REGION Network 7: GlueCalibratonMode Manual Mode Reset Test
   RUNG wire#powerrail
      Contact( "Station_Sys".Manual.Mode )
      Contact( "GluingControl".GlueCalibratonMode )
      Contact( "GluingControl".Control.ManualTest_X )
      Contact( "IAI_DeviceCtl".IAIServo[2].Point[1].Achieve )
      Contact( "IAI_DeviceCtl".IAIServo[1].Point[1].Achieve )
      Contact( "IAI_DeviceCtl".IAIServo[3].Point[1].Achieve )
      { S7_Templates := "time_type := LTime" } "GluingControl".TON[1].TONR(r := wire#w2, pt := LT#10.7S, et =>)
   END_RUNG
   RUNG wire#powerrail
      Contact( "GluingControl".GlueCalibratonMode )
      wire#w1
      P_Trig( "GluingControl".P[1] )
   END_RUNG wire#w2
   RUNG wire#powerrail
      I_Contact( "Station_Sys".Manual.Mode )
   END_RUNG wire#w1
   RUNG wire#powerrail
      { S7_Templates := "SrcType := LTime" } EQ_Contact(in1 := "GluingControl".TON[1].ET, in2 := LT#10.7S)
      R_Coil( "GluingControl".Control.ManualTest_X )
      R_Coil( "GluingControl".GlueCalibratonMode )
   END_RUNG
   // the same network as SCL:
   #_w1 := "GluingControl".GlueCalibratonMode OR NOT "Station_Sys".Manual.Mode;
   #_w2 := #_w1 AND NOT "GluingControl".P[1];   // rising edge
   "GluingControl".P[1] := #_w1;
   "GluingControl".TON[1].TONR(IN := "Station_Sys".Manual.Mode AND "GluingControl".GlueCalibratonMode AND "GluingControl".Control.ManualTest_X AND "IAI_DeviceCtl".IAIServo[2].Point[1].Achieve AND "IAI_DeviceCtl".IAIServo[1].Point[1].Achieve AND "IAI_DeviceCtl".IAIServo[3].Point[1].Achieve,
                           R := #_w2,
                           PT := LT#10.7S);
   IF "GluingControl".TON[1].ET = LT#10.7S THEN
       "GluingControl".Control.ManualTest_X := FALSE;
       "GluingControl".GlueCalibratonMode := FALSE;
   END_IF;
END_REGION
END_FUNCTION

FUNCTION "Pallet_NG" : Void   // FC2900, LAD
{ S7_Optimized_Access := 'TRUE' }
// stored: AutoNumber false, SetENOAutomatically false
   VAR_INPUT
      iSysMode : "RCS_SysComInterface_V1";
   END_VAR
BEGIN

REGION Network 1 (SCL): NG BOXES MAIN FUNCTION BLOCK
   "NG_BOXES_DB"(
                 in_Permission_to_Open :=
                 // in manual mode always
                 #iSysMode.ManualMode OR
                 // 
                 (
                 // all 3 robots are in safe step and have no job / no task running
                 "ST10_Flow5_FRobot_1_iDB"."Open NG BOX REQUESTED?".X AND
                 "ST10_Flow8_FRobot_2_iDB"."Open NG BOX REQUESTED?".X AND
                 "ST10_Flow15_FRobot_3_iDB"."Open NG BOX REQUESTED?".X
                 ) OR "Robot_DB".NG_box_open_flag_during_auto
                 );
END_REGION
END_FUNCTION

FUNCTION_BLOCK "NG_BOXES"   // FB3, SCL
{ S7_Optimized_Access := 'TRUE' }
// stored: MemoryReserve 1000, SetENOAutomatically false
   VAR_INPUT
      in_Permission_to_Open : Bool;
   END_VAR
   VAR_OUTPUT
      out_Request_to_open : Bool;
   END_VAR
   VAR
      Box_Loading { S7_SetPoint := 'True'} : "FB_NG_Box_Control";
      Box_Unloading { S7_SetPoint := 'True'} : "FB_NG_Box_Control";
      TempSensors : Array[1..15] of Bool;
   END_VAR
BEGIN
   // ==========================================================================
   // BOX 1: LOADING – MACHINE LOADING SIDE                                   // EN: Loading side of machine (material IN)
   //                                                                          // CN: 机器上料侧（物料进入机器）
   //                                                                          // SK: Nakladacia / vstupná strana stroja
   // ==========================================================================
   #TempSensors[1] := "iE1-UnloadingShaftPressNG_1";   // EN: NG shaft press pos 1   // CN: 轴压装NG位置1   // SK: NG lis hriadeľa poz.1
   #TempSensors[2] := "iE1-UnloadingShaftPressNG_2";   // EN: NG shaft press pos 2   // CN: 轴压装NG位置2   // SK: NG lis hriadeľa poz.2
   #TempSensors[3] := "iE1-UnloadingShaftPressNG_3";   // EN: NG shaft press pos 3   // CN: 轴压装NG位置3   // SK: NG lis hriadeľa poz.3
   #TempSensors[4] := "iE1-UnloadingShaftPressNG_4";   // EN: NG shaft press pos 4   // CN: 轴压装NG位置4   // SK: NG lis hriadeľa poz.4
   #TempSensors[5] := "iE1-UnloadingShaftPressNG_5";   // EN: NG shaft press pos 5   // CN: 轴压装NG位置5   // SK: NG lis hriadeľa poz.5
   #TempSensors[6] := "iE1-UnloadingShaftScanNG_1";    // EN: NG shaft scan pos 1    // CN: 轴扫描NG位置1   // SK: NG sken hriadeľa 1
   #TempSensors[7] := "iE1-UnloadingShaftScanNG_2";    // EN: NG shaft scan pos 2    // CN: 轴扫描NG位置2   // SK: NG sken hriadeľa 2
   #TempSensors[8] := "iE1-UnloadingShaftScanNG_3";    // EN: NG shaft scan pos 3    // CN: 轴扫描NG位置3   // SK: NG sken hriadeľa 3
   #TempSensors[9] := "iE1-UnloadingShaftScanNG_4";    // EN: NG shaft scan pos 4    // CN: 轴扫描NG位置4   // SK: NG sken hriadeľa 4
   #TempSensors[10] := "iE1-UnloadingShaftScanNG_5";    // EN: NG shaft scan pos 5    // CN: 轴扫描NG位置5   // SK: NG sken hriadeľa 5
   #TempSensors[11] := "iE1-UnloadingRingScanNG_1";     // EN: NG ring scan pos 1     // CN: 环扫描NG位置1   // SK: NG sken krúžku 1
   #TempSensors[12] := "iE1-UnloadingRingScanNG_2";     // EN: NG ring scan pos 2     // CN: 环扫描NG位置2   // SK: NG sken krúžku 2
   #TempSensors[13] := "iE1-UnloadingRingScanNG_3";     // EN: NG ring scan pos 3     // CN: 环扫描NG位置3   // SK: NG sken krúžku 3
   #TempSensors[14] := "iE1-UnloadingRingScanNG_4";     // EN: NG ring scan pos 4     // CN: 环扫描NG位置4   // SK: NG sken krúžku 4
   #TempSensors[15] := "iE1-UnloadingRingScanNG_5";     // EN: NG ring scan pos 5     // CN: 环扫描NG位置5   // SK: NG sken krúžku 5

   #Box_Loading(
                Button        := "iNG_Button1",                     // EN: Operator button (loading side)   // CN: 上料侧操作按钮   // SK: Tlačidlo obsluhy – loading
                MagnetSensor  := "iE-NG-01Detection",               // EN: Door closed sensor                // CN: 门关闭传感器     // SK: Snímač zatvorenia dverí
                LockedFB      := NOT "iE-NG-01 Safety Gate_UnLock", // EN: Lock feedback (locked)             // CN: 锁定反馈         // SK: Spätná väzba – zamknuté
                UnlockedFB    := "iE-NG-01 Safety Gate_UnLock",     // EN: Lock feedback (unlocked)           // CN: 解锁反馈         // SK: Spätná väzba – odomknuté
                AtSafePoint   := #in_Permission_to_Open,            // EN: Sequence at safe point (Step 111)  // CN: 序列在安全步骤   // SK: Sekvencia v bezpečnom kroku
                Sensors       := #TempSensors,
                UnlockCmd     => "ST10_NGGate1_DB"."sSafetyGate UnlockRequest", // EN: Unlock command // CN: 解锁命令 // SK: Príkaz na odomknutie
                LockCmd       => "ST10_NGGate1_DB"."sSafetyGate LockRequest",   // EN: Lock command   // CN: 上锁命令 // SK: Príkaz na zamknutie
                CylinderOpen  => "oE-NG-01NGLocationCylinderToHP",   // EN: Cylinder open (home)  // CN: 气缸打开 // SK: Otvoriť valec
                CylinderClose => "oE-NG-01NGLocationCylinderToWP",   // EN: Cylinder close (work) // CN: 气缸关闭 // SK: Zavrieť valec
                ButtonLight => "oNG_Button1"   ,                    // E,N: Button lamp           // CN: 按钮灯   // SK: Svetlo tlačidla
                Ready_1 => "AutoProcessControl".NG_1.Robot1PutPrimit_1   ,         // Status pro robota: Řada 1 (1-5) má místo // 机器人状态：第1排（1-5）有空位
                Ready_2 => "AutoProcessControl".NG_1.Robot1PutPrimit_2,
                Ready_3 => "AutoProcessControl".NG_1.Robot1PutPrimit_3

   );

   // ==========================================================================
   // BOX 2: UNLOADING – MACHINE UNLOADING SIDE                                // EN: Unloading side of machine (material OUT)
   //                                                                          // CN: 机器下料侧（物料离开机器）
   //                                                                          // SK: Vykladacia / výstupná strana stroja
   // ==========================================================================
   #TempSensors[1] := "iE2-UnloadingPressNG_1";          // EN: NG press pos 1   // CN: 压装NG位置1   // SK: NG lis poz.1
   #TempSensors[2] := "iE2-UnloadingPressNG_2";          // EN: NG press pos 2   // CN: 压装NG位置2   // SK: NG lis poz.2
   #TempSensors[3] := "iE2-UnloadingPressNG_3";          // EN: NG press pos 3   // CN: 压装NG位置3   // SK: NG lis poz.3
   #TempSensors[4] := "iE2-UnloadingPressNG_4";          // EN: NG press pos 4   // CN: 压装NG位置4   // SK: NG lis poz.4
   #TempSensors[5] := "iE2-UnloadingPressNG_5";          // EN: NG press pos 5   // CN: 压装NG位置5   // SK: NG lis poz.5
   #TempSensors[6] := "iE2-UnloadingMagentScanNG_1";     // EN: NG magnet scan 1 // CN: 磁体扫描NG1   // SK: NG magnet sken 1
   #TempSensors[7] := "iE2-UnloadingMagentScanNG_2";     // EN: NG magnet scan 2 // CN: 磁体扫描NG2   // SK: NG magnet sken 2
   #TempSensors[8] := "iE2-UnloadingMagentScanNG_3";     // EN: NG magnet scan 3 // CN: 磁体扫描NG3   // SK: NG magnet sken 3
   #TempSensors[9] := "iE2-UnloadingMagentScanNG_4";     // EN: NG magnet scan 4 // CN: 磁体扫描NG4   // SK: NG magnet sken 4
   #TempSensors[10] := "iE2-UnloadingMagentScanNG_5";     // EN: NG magnet scan 5 // CN: 磁体扫描NG5   // SK: NG magnet sken 5
   #TempSensors[11] := "iE2-UnloadingRingScanNG_1";       // EN: NG ring scan 1   // CN: 环扫描NG1     // SK: NG sken krúžku 1
   #TempSensors[12] := "iE2-UnloadingRingScanNG_2";       // EN: NG ring scan 2   // CN: 环扫描NG2     // SK: NG sken krúžku 2
   #TempSensors[13] := "iE2-UnloadingRingScanNG_3";       // EN: NG ring scan 3   // CN: 环扫描NG3     // SK: NG sken krúžku 3
   #TempSensors[14] := "iE2-UnloadingRingScanNG_4";       // EN: NG ring scan 4   // CN: 环扫描NG4     // SK: NG sken krúžku 4
   #TempSensors[15] := "iE2-UnloadingRingScanNG_5";       // EN: NG ring scan 5   // CN: 环扫描NG5     // SK: NG sken krúžku 5

   #Box_Unloading(
                  Button        := "iNG_Button2",                     // EN: Operator button (unloading side) // CN: 下料侧操作按钮 // SK: Tlačidlo obsluhy – unloading
                  MagnetSensor  := "iE-NG-02Detection",               // EN: Door closed sensor               // CN: 门关闭传感器   // SK: Snímač zatvorenia dverí
                  LockedFB      := NOT "iE-NG-02 Safety Gate_UnLock", // EN: Lock feedback (locked)            // CN: 锁定反馈       // SK: Spätná väzba – zamknuté
                  UnlockedFB    := "iE-NG-02 Safety Gate_UnLock",     // EN: Lock feedback (unlocked)          // CN: 解锁反馈       // SK: Spätná väzba – odomknuté
                  AtSafePoint   := #in_Permission_to_Open,
                  Sensors       := #TempSensors,
                  UnlockCmd     => "ST10_NGGate2_DB"."sSafetyGate UnlockRequest",
                  LockCmd       => "ST10_NGGate2_DB"."sSafetyGate LockRequest",
                  CylinderOpen  => "oE-NG-02NGLocationCylinderToHP",
                  CylinderClose => "oE-NG-02NGLocationCylinderToWP",
                  ButtonLight   => "oNG_Button2",
                  Ready_1 => "AutoProcessControl".NG_2.Robot3PutPrimit_1   ,         // Status pro robota: Řada 1 (1-5) má místo // 机器人状态：第1排（1-5）有空位
                  Ready_2 => "AutoProcessControl".NG_2.Robot3PutPrimit_2,
                  Ready_3 => "AutoProcessControl".NG_2.Robot3PutPrimit_3
   );

   // EN: Request pause of main sequence if any side requests opening
   // CN: 任一侧请求开门时，请求暂停主序列
   // SK: Požiadavka na pauzu hlavnej sekvencie, ak ktorákoľvek strana žiada otvorenie
   #out_Request_to_open := #Box_Loading.PauseReq OR #Box_Unloading.PauseReq;
END_FUNCTION_BLOCK

FUNCTION_BLOCK "FB_NG_Box_Control"   // FB5, SCL
{ S7_Optimized_Access := 'TRUE' }
// stored: MemoryReserve 1000, SetENOAutomatically false
   VAR_INPUT
      Button : Bool;
      MagnetSensor : Bool;
      LockedFB : Bool;
      UnlockedFB : Bool;
      AtSafePoint : Bool;
      Sensors : Array[1..15] of Bool;
   END_VAR
   VAR_OUTPUT
      PauseReq : Bool;
      UnlockCmd : Bool;
      LockCmd : Bool;
      CylinderOpen : Bool;
      CylinderClose : Bool;
      ButtonLight : Bool;
      Ready_1 : Bool;
      Ready_2 : Bool;
      Ready_3 : Bool;
      OpenFlag : Bool;
   END_VAR
   VAR
      State : Int := 99;
      BlinkTimer { S7_SetPoint := 'True'} : TON_TIME;
      BlinkBit : Bool;
      i : Int;
      buttontriggered { S7_SetPoint := 'True'} : R_TRIG;
      c : Int;
   END_VAR
BEGIN
   // 1. POSITION CHECK (Ready_1..3) - TRUE = at least one position in the row is FREE
   // 1. KONTROLA POZÍCIÍ – TRUE = aspoň jedna pozícia v rade je VOĽNÁ
   // 1. 位置检测 – TRUE = 该行中至少有一个位置是空的

   // LINE #1  .... 5 POSITIONS
   // EN: Line 1 checks sensors 1–5 (row 1)
   // SK: Riadok 1 kontroluje senzory 1–5 (riadok 1)
   // CN: 第1行检测传感器1–5（第1排）
   #Ready_1 := FALSE;
   FOR #i := 1 TO 5 DO
     IF NOT #Sensors[#i] THEN
       #Ready_1 := TRUE;
     END_IF;
   END_FOR;

   // LINE #2  .... 5 POSITIONS
   // EN: Line 2 checks sensors 6–10 (row 2)
   // SK: Riadok 2 kontroluje senzory 6–10 (riadok 2)
   // CN: 第2行检测传感器6–10（第2排）
   #Ready_2 := FALSE;
   FOR #i := 6 TO 10 DO
     IF NOT #Sensors[#i] THEN
       #Ready_2 := TRUE;
     END_IF;
   END_FOR;

   // LINE #3  .... 5 POSITIONS
   // EN: Line 3 checks sensors 11–15 (row 3)
   // SK: Riadok 3 kontroluje senzory 11–15 (riadok 3)
   // CN: 第3行检测传感器11–15（第3排）
   #Ready_3 := FALSE;
   FOR #i := 11 TO 15 DO
     IF NOT #Sensors[#i] THEN
       #Ready_3 := TRUE;
     END_IF;
   END_FOR;


   // 2. BLINKING / BUTTON FEEDBACK
   // EN: Blink signal taken from system clock (0.4s)
   // SK: Blikanie je odvodené zo systémového hodinového bitu (0,4 s)
   // CN: 闪烁信号来自系统时钟位（0.4秒）
   #BlinkBit := "ClockMemory0.4s";

   // EN: Rising-edge detection of the button
   // SK: Detekcia nábežnej hrany tlačidla
   // CN: 按钮上升沿检测
   #buttontriggered(CLK := #Button);


   // 3. DOOR STATE MACHINE
   // EN: Main state machine controlling door, lock and cylinder
   // SK: Hlavný stavový automat pre dvere, zámok a valec
   // CN: 门、锁和气缸的主状态机
   CASE #State OF

     99: // INITIALIZATION
       // EN: Decision after PLC start
       // SK: Rozhodnutie po štarte PLC
       // CN: PLC 启动后的状态判断
       IF #MagnetSensor AND #LockedFB THEN
         #State := 0;   // EN: Closed & locked → IDLE
         // SK: Zavreté a zamknuté → IDLE
         // CN: 已关闭并锁定 → 空闲状态
       ELSIF #MagnetSensor AND NOT #LockedFB THEN
         #State := 40;  // EN: Closed but unlocked → wait for confirmation
         // SK: Zavreté, ale odomknuté → čakať na potvrdenie
         // CN: 门已关但未上锁 → 等待确认
       ELSE
         #State := 30;  // EN: Door physically open → OPEN state
         // SK: Dvere fyzicky otvorené → OPEN stav
         // CN: 门处于打开状态 → OPEN
       END_IF;

     0:  // IDLE
       // EN: Normal operation, sequence running
       // SK: Normálna prevádzka, sekvencia beží
       // CN: 正常运行，工序执行中
       #PauseReq := FALSE;
       #UnlockCmd := FALSE;
       #LockCmd := TRUE;
       #CylinderOpen := FALSE;
       #CylinderClose := TRUE;
       #ButtonLight := TRUE;
       #OpenFlag := FALSE;
       IF #buttontriggered.Q THEN
         #State := 10;
       END_IF;

     10: // REQUEST
       // EN: Button pressed, waiting for safe point (Step 111)
       // SK: Tlačidlo stlačené, čaká sa na bezpečný bod (Krok 111)
       // CN: 按钮按下，等待安全点（步骤111）
       #PauseReq := TRUE;
       #ButtonLight := #BlinkBit;
       IF #AtSafePoint THEN
         #State := 20;
       END_IF;

     20: // SAFE
       // EN: Sequence stopped, unlocking door and opening cylinder
       // SK: Sekvencia stojí, odomykáme dvere a otvárame valec
       // CN: 工序停止，解锁门并打开气缸
       #PauseReq := TRUE;
       #UnlockCmd := TRUE;
       #LockCmd := FALSE;
       #ButtonLight := #BlinkBit;
       IF #UnlockedFB THEN
         #CylinderOpen := TRUE;
         #CylinderClose := FALSE;
         #State := 30;
       END_IF;

     30: // OPEN
       // EN: Door open, operator access
       // SK: Dvere otvorené, obsluha má prístup
       // CN: 门已打开，操作员可进入
       #PauseReq := TRUE;
       #ButtonLight := FALSE;
       #OpenFlag := TRUE;
       #UnlockCmd := TRUE;
       #LockCmd := FALSE;
       #CylinderOpen := TRUE;
       #CylinderClose := FALSE;
       IF #MagnetSensor THEN
         #State := 40;
       END_IF;

     40: // CONFIRM
       // EN: Door closed, waiting for operator confirmation
       // SK: Dvere zatvorené, čaká sa na potvrdenie obsluhou
       // CN: 门已关闭，等待人工确认
       #PauseReq := TRUE;
       #ButtonLight := #BlinkBit;
       #OpenFlag := TRUE;
       #UnlockCmd := TRUE;
       #LockCmd := FALSE;
       #CylinderOpen := TRUE;
       #CylinderClose := FALSE;
       IF NOT #MagnetSensor THEN
         #State := 30;
       ELSIF #buttontriggered.Q THEN
         #State := 50;
       END_IF;

     50: // LOCKING
       // EN: Locking door and returning cylinder
       // SK: Zamykáme dvere a vraciame valec
       // CN: 锁门并回收气缸
       #PauseReq := TRUE;
       #CylinderOpen := FALSE;
       #CylinderClose := TRUE;
       #UnlockCmd := FALSE;
       #LockCmd := TRUE;
       IF #LockedFB THEN
         #PauseReq := FALSE; // EN: Release Step 111, sequence continues
         // SK: Uvoľní sa Krok 111, sekvencia pokračuje
         // CN: 释放步骤111，工序继续
         #State := 0;
       END_IF;

   END_CASE;


   // EN: Test lamp function from system diagnostics
   // SK: Testovacia funkcia lampy zo systémovej diagnostiky
   // CN: 系统诊断用的灯测试功能
   IF "Station_Sys".Cmd.TestLamp THEN
     #ButtonLight := TRUE;
   END_IF;
END_FUNCTION_BLOCK

FUNCTION "MES" : Void   // FC500, LAD
{ S7_Optimized_Access := 'TRUE' }
// stored: AutoNumber false, SetENOAutomatically false
   VAR_TEMP
      YEAR : Int;
      MONTH : Int;
      DAY : Int;
      HH : Int;
      MM : Int;
      SS : Int;
      RET1 : Int;
      RET2 : Int;
      P : Array[0..10] of Bool;
   END_VAR
   VAR_TEMP   // added for the SCL form of the ladder/FBD networks
      _w1 : Bool;
      _w2 : Bool;
   END_VAR
BEGIN

REGION Network 2: 自动复位测试 / Automatic reset test
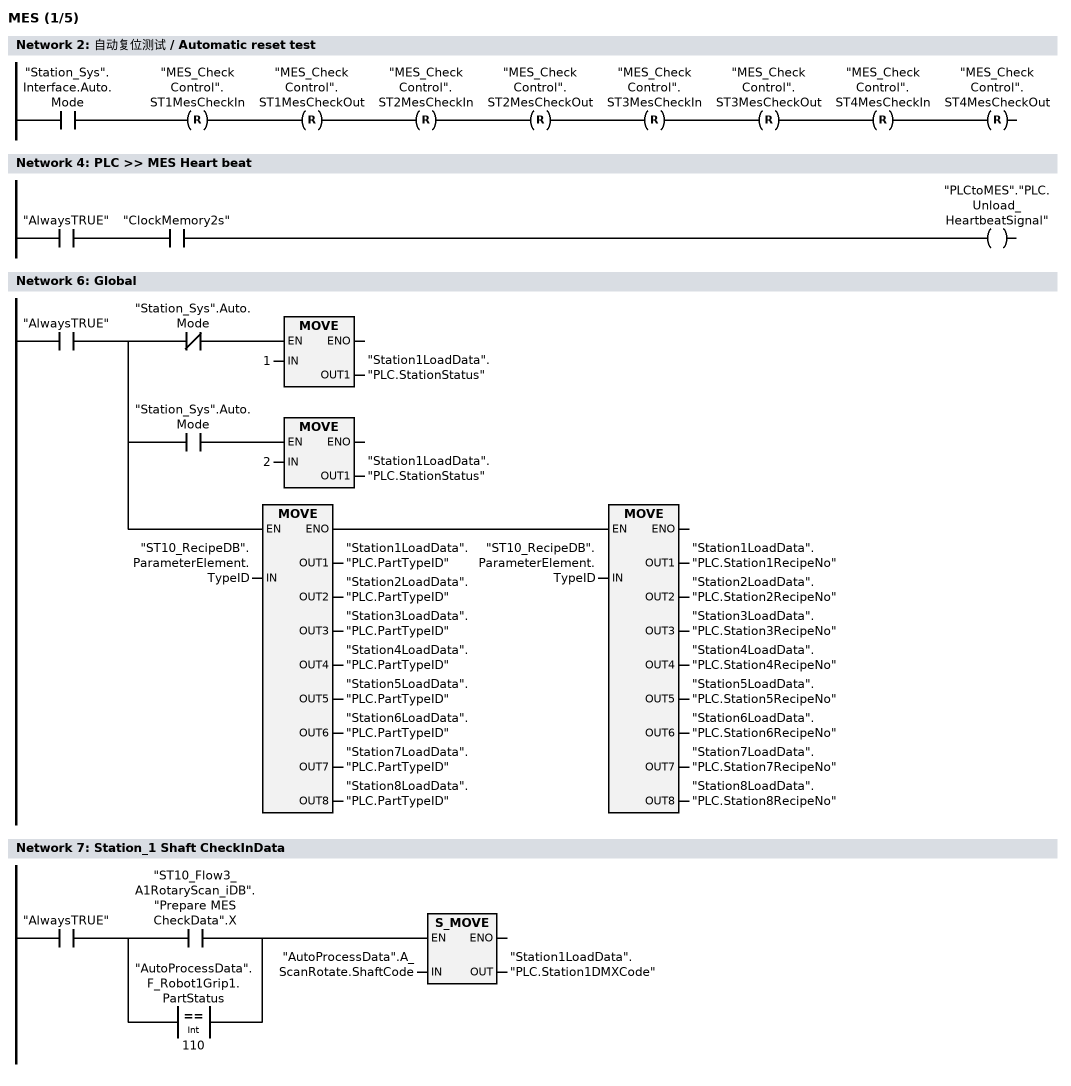
   RUNG wire#powerrail
      Contact( "Station_Sys".Interface.Auto.Mode )
      R_Coil( "MES_CheckControl".ST1MesCheckIn )
      R_Coil( "MES_CheckControl".ST1MesCheckOut )
      R_Coil( "MES_CheckControl".ST2MesCheckIn )
      R_Coil( "MES_CheckControl".ST2MesCheckOut )
      R_Coil( "MES_CheckControl".ST3MesCheckIn )
      R_Coil( "MES_CheckControl".ST3MesCheckOut )
      R_Coil( "MES_CheckControl".ST4MesCheckIn )
      R_Coil( "MES_CheckControl".ST4MesCheckOut )
   END_RUNG
   // the same network as SCL:
   IF "Station_Sys".Interface.Auto.Mode THEN
       "MES_CheckControl".ST1MesCheckIn := FALSE;
       "MES_CheckControl".ST1MesCheckOut := FALSE;
       "MES_CheckControl".ST2MesCheckIn := FALSE;
       "MES_CheckControl".ST2MesCheckOut := FALSE;
       "MES_CheckControl".ST3MesCheckIn := FALSE;
       "MES_CheckControl".ST3MesCheckOut := FALSE;
       "MES_CheckControl".ST4MesCheckIn := FALSE;
       "MES_CheckControl".ST4MesCheckOut := FALSE;
   END_IF;
END_REGION

NETWORK
TITLE = PLC系统时间转换 / PLC system time conversion
//########提取PLC当前日期
      L     %DB3000.DBB18;
      BTI;
      T     #YEAR;
      L     %DB3000.DBB19;
      BTI;
      T     #MONTH;
      L     %DB3000.DBB20;
      BTI;
      T     #DAY;
      L     %DB3000.DBB21;
      BTI;
      T     #HH;
      L     %DB3000.DBB22;
      BTI;
      T     #MM;
      L     %DB3000.DBB23;
      BTI;
      T     #SS;


//########将日期转化成字符
      CALL  "DT-Chars", "DT-Chars_DB"
      ( YEAR                := #YEAR,
        MONTH               := #MONTH,
        DAY                 := #DAY,
        HH                  := #HH,
        MM                  := #MM,
        SS                  := #SS,
        Year_Byte1          := ,
        Year_Byte2          := ,
        Month_Byte1         := ,
        Month_Byte2         := ,
        Days_Byte1          := ,
        Days_Byte2          := ,
        HH_Byte1            := ,
        HH_Byte2            := ,
        MM_Byte1            := ,
        MM_Byte2            := ,
        SS_Byte1            := ,
        SS_Byte2            := ,
        CalculateDays_Byte1 := ,
        CalculateDays_Byte2 := ,
        CalculateDays_Byte3 := ,
        Error_Code          := ,
        Year_Byte3          := ,
        Year_Byte4          := ,
        Month_Byte3         := ,
        Month_Byte4         := ,
        Days_Byte3          := ,
        Days_Byte4          := ,
        HH_Byte3            := ,
        HH_Byte4            := ,
        MM_Byte3            := ,
        MM_Byte4            := ,
        SS_Byte3            := ,
        SS_Byte4            := ,
        CalculateDays_Byte4 := ,
        CalculateDays_Byte5 := ,
        CalculateDays_Byte6 := ,
        OTimeStr            := 
      );




REGION Network 4: PLC >> MES Heart beat
   RUNG wire#powerrail
      Contact( "AlwaysTRUE" )
      Contact( "ClockMemory2s" )
      Coil( "PLCtoMES"."PLC.Unload_HeartbeatSignal" )
   END_RUNG
   // the same network as SCL:
   "PLCtoMES"."PLC.Unload_HeartbeatSignal" := "AlwaysTRUE" AND "ClockMemory2s";
END_REGION

REGION Network 6: Global
   RUNG wire#powerrail
      Contact( "AlwaysTRUE" )
      wire#w1
      I_Contact( "Station_Sys".Auto.Mode )
      Move(in := 1, out1 => "Station1LoadData"."PLC.StationStatus")
   END_RUNG
   RUNG wire#w1
      Contact( "Station_Sys".Auto.Mode )
      Move(in := 2, out1 => "Station1LoadData"."PLC.StationStatus")
   END_RUNG
   RUNG wire#w1
      Move(in := "ST10_RecipeDB".ParameterElement.TypeID, out1 => "Station1LoadData"."PLC.PartTypeID", out2 => "Station2LoadData"."PLC.PartTypeID", out3 => "Station3LoadData"."PLC.PartTypeID", out4 => "Station4LoadData"."PLC.PartTypeID", out5 => "Station5LoadData"."PLC.PartTypeID", out6 => "Station6LoadData"."PLC.PartTypeID", out7 => "Station7LoadData"."PLC.PartTypeID", out8 => "Station8LoadData"."PLC.PartTypeID")
      Move(in := "ST10_RecipeDB".ParameterElement.TypeID, out1 => "Station1LoadData"."PLC.Station1RecipeNo", out2 => "Station2LoadData"."PLC.Station2RecipeNo", out3 => "Station3LoadData"."PLC.Station3RecipeNo", out4 => "Station4LoadData"."PLC.Station4RecipeNo", out5 => "Station5LoadData"."PLC.Station5RecipeNo", out6 => "Station6LoadData"."PLC.Station6RecipeNo", out7 => "Station7LoadData"."PLC.Station7RecipeNo", out8 => "Station8LoadData"."PLC.Station8RecipeNo")
   END_RUNG
   // the same network as SCL:
   IF "AlwaysTRUE" AND NOT "Station_Sys".Auto.Mode THEN "Station1LoadData"."PLC.StationStatus" := 1; END_IF;
   IF "AlwaysTRUE" AND "Station_Sys".Auto.Mode THEN "Station1LoadData"."PLC.StationStatus" := 2; END_IF;
   IF "AlwaysTRUE" THEN
       "Station1LoadData"."PLC.PartTypeID" := "ST10_RecipeDB".ParameterElement.TypeID;
       "Station2LoadData"."PLC.PartTypeID" := "ST10_RecipeDB".ParameterElement.TypeID;
       "Station3LoadData"."PLC.PartTypeID" := "ST10_RecipeDB".ParameterElement.TypeID;
       "Station4LoadData"."PLC.PartTypeID" := "ST10_RecipeDB".ParameterElement.TypeID;
       "Station5LoadData"."PLC.PartTypeID" := "ST10_RecipeDB".ParameterElement.TypeID;
       "Station6LoadData"."PLC.PartTypeID" := "ST10_RecipeDB".ParameterElement.TypeID;
       "Station7LoadData"."PLC.PartTypeID" := "ST10_RecipeDB".ParameterElement.TypeID;
       "Station8LoadData"."PLC.PartTypeID" := "ST10_RecipeDB".ParameterElement.TypeID;
       "Station1LoadData"."PLC.Station1RecipeNo" := "ST10_RecipeDB".ParameterElement.TypeID;
       "Station2LoadData"."PLC.Station2RecipeNo" := "ST10_RecipeDB".ParameterElement.TypeID;
       "Station3LoadData"."PLC.Station3RecipeNo" := "ST10_RecipeDB".ParameterElement.TypeID;
       "Station4LoadData"."PLC.Station4RecipeNo" := "ST10_RecipeDB".ParameterElement.TypeID;
       "Station5LoadData"."PLC.Station5RecipeNo" := "ST10_RecipeDB".ParameterElement.TypeID;
       "Station6LoadData"."PLC.Station6RecipeNo" := "ST10_RecipeDB".ParameterElement.TypeID;
       "Station7LoadData"."PLC.Station7RecipeNo" := "ST10_RecipeDB".ParameterElement.TypeID;
       "Station8LoadData"."PLC.Station8RecipeNo" := "ST10_RecipeDB".ParameterElement.TypeID;
   END_IF;
END_REGION

REGION Network 7: Station_1 Shaft CheckInData
   RUNG wire#powerrail
      Contact( "AlwaysTRUE" )
      wire#w1
      Contact( "ST10_Flow3_A1RotaryScan_iDB"."Prepare MES CheckData".X )
      wire#w2
      S_Move(in := "AutoProcessData".A_ScanRotate.ShaftCode, out => "Station1LoadData"."PLC.Station1DMXCode")
   END_RUNG
   RUNG wire#w1
      { S7_Templates := "SrcType := Int" } EQ_Contact(in1 := "AutoProcessData".F_Robot1Grip1.PartStatus, in2 := 110)
   END_RUNG wire#w2
   // the same network as SCL:
   IF "AlwaysTRUE" AND ("ST10_Flow3_A1RotaryScan_iDB"."Prepare MES CheckData".X OR ("AutoProcessData".F_Robot1Grip1.PartStatus = 110)) THEN
       "Station1LoadData"."PLC.Station1DMXCode" := "AutoProcessData".A_ScanRotate.ShaftCode;
   END_IF;
END_REGION

REGION Network 8: Station_1 Shaft CheckResultData
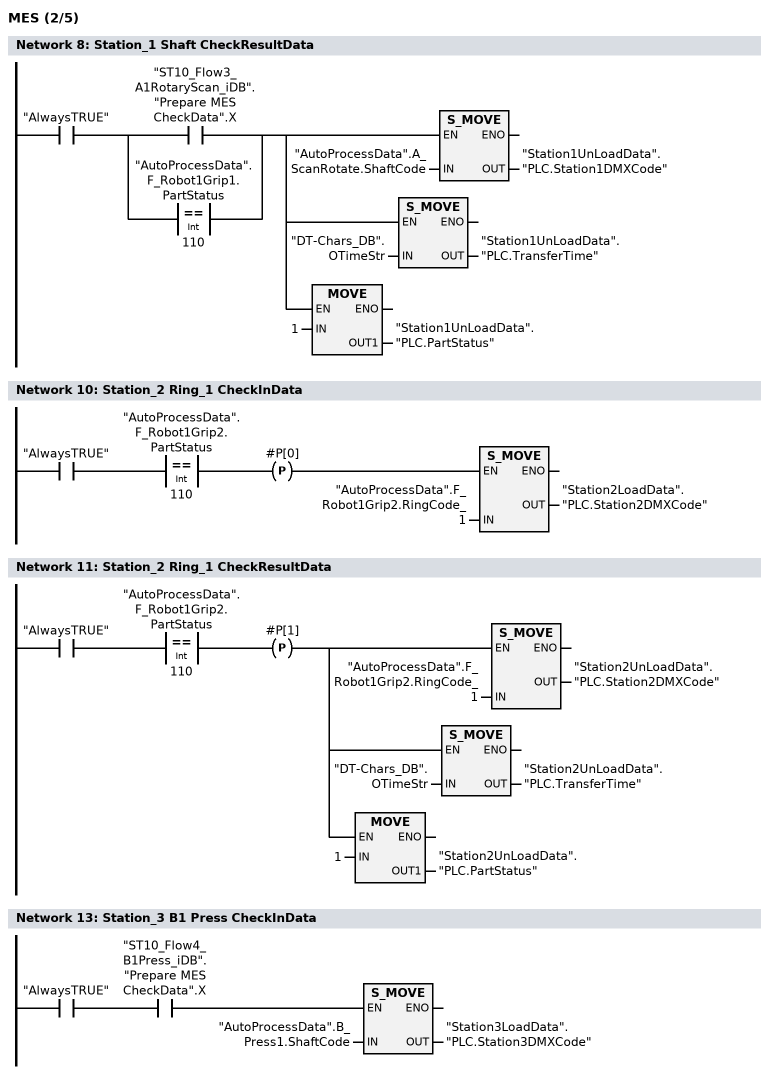
   RUNG wire#powerrail
      Contact( "AlwaysTRUE" )
      wire#w1
      Contact( "ST10_Flow3_A1RotaryScan_iDB"."Prepare MES CheckData".X )
      wire#w2
      S_Move(in := "AutoProcessData".A_ScanRotate.ShaftCode, out => "Station1UnLoadData"."PLC.Station1DMXCode")
   END_RUNG
   RUNG wire#w1
      { S7_Templates := "SrcType := Int" } EQ_Contact(in1 := "AutoProcessData".F_Robot1Grip1.PartStatus, in2 := 110)
   END_RUNG wire#w2
   RUNG wire#w2
      S_Move(in := "DT-Chars_DB".OTimeStr, out => "Station1UnLoadData"."PLC.TransferTime")
   END_RUNG
   RUNG wire#w2
      Move(in := 1, out1 => "Station1UnLoadData"."PLC.PartStatus")
   END_RUNG
   // the same network as SCL:
   IF "AlwaysTRUE" AND ("ST10_Flow3_A1RotaryScan_iDB"."Prepare MES CheckData".X OR ("AutoProcessData".F_Robot1Grip1.PartStatus = 110)) THEN
       "Station1UnLoadData"."PLC.Station1DMXCode" := "AutoProcessData".A_ScanRotate.ShaftCode;
       "Station1UnLoadData"."PLC.TransferTime" := "DT-Chars_DB".OTimeStr;
       "Station1UnLoadData"."PLC.PartStatus" := 1;
   END_IF;
END_REGION

REGION Network 10: Station_2 Ring_1 CheckInData
   RUNG wire#powerrail
      Contact( "AlwaysTRUE" )
      { S7_Templates := "SrcType := Int" } EQ_Contact(in1 := "AutoProcessData".F_Robot1Grip2.PartStatus, in2 := 110)
      P_Trig( #P[0] )
      S_Move(in := "AutoProcessData".F_Robot1Grip2.RingCode_1, out => "Station2LoadData"."PLC.Station2DMXCode")
   END_RUNG
   // the same network as SCL:
   #_w1 := "AlwaysTRUE" AND ("AutoProcessData".F_Robot1Grip2.PartStatus = 110);
   #_w2 := #_w1 AND NOT #P[0];   // rising edge
   #P[0] := #_w1;
   IF #_w2 THEN
       "Station2LoadData"."PLC.Station2DMXCode" := "AutoProcessData".F_Robot1Grip2.RingCode_1;
   END_IF;
END_REGION

REGION Network 11: Station_2 Ring_1 CheckResultData
   RUNG wire#powerrail
      Contact( "AlwaysTRUE" )
      { S7_Templates := "SrcType := Int" } EQ_Contact(in1 := "AutoProcessData".F_Robot1Grip2.PartStatus, in2 := 110)
      P_Trig( #P[1] )
      wire#w1
      S_Move(in := "AutoProcessData".F_Robot1Grip2.RingCode_1, out => "Station2UnLoadData"."PLC.Station2DMXCode")
   END_RUNG
   RUNG wire#w1
      S_Move(in := "DT-Chars_DB".OTimeStr, out => "Station2UnLoadData"."PLC.TransferTime")
   END_RUNG
   RUNG wire#w1
      Move(in := 1, out1 => "Station2UnLoadData"."PLC.PartStatus")
   END_RUNG
   // the same network as SCL:
   #_w1 := "AlwaysTRUE" AND ("AutoProcessData".F_Robot1Grip2.PartStatus = 110);
   #_w2 := #_w1 AND NOT #P[1];   // rising edge
   #P[1] := #_w1;
   IF #_w2 THEN
       "Station2UnLoadData"."PLC.Station2DMXCode" := "AutoProcessData".F_Robot1Grip2.RingCode_1;
       "Station2UnLoadData"."PLC.TransferTime" := "DT-Chars_DB".OTimeStr;
       "Station2UnLoadData"."PLC.PartStatus" := 1;
   END_IF;
END_REGION

REGION Network 13: Station_3 B1 Press CheckInData
   RUNG wire#powerrail
      Contact( "AlwaysTRUE" )
      Contact( "ST10_Flow4_B1Press_iDB"."Prepare MES CheckData".X )
      S_Move(in := "AutoProcessData".B_Press1.ShaftCode, out => "Station3LoadData"."PLC.Station3DMXCode")
   END_RUNG
   // the same network as SCL:
   IF "AlwaysTRUE" AND "ST10_Flow4_B1Press_iDB"."Prepare MES CheckData".X THEN
       "Station3LoadData"."PLC.Station3DMXCode" := "AutoProcessData".B_Press1.ShaftCode;
   END_IF;
END_REGION

REGION Network 14: Station_3 B1 Press CheckResultData
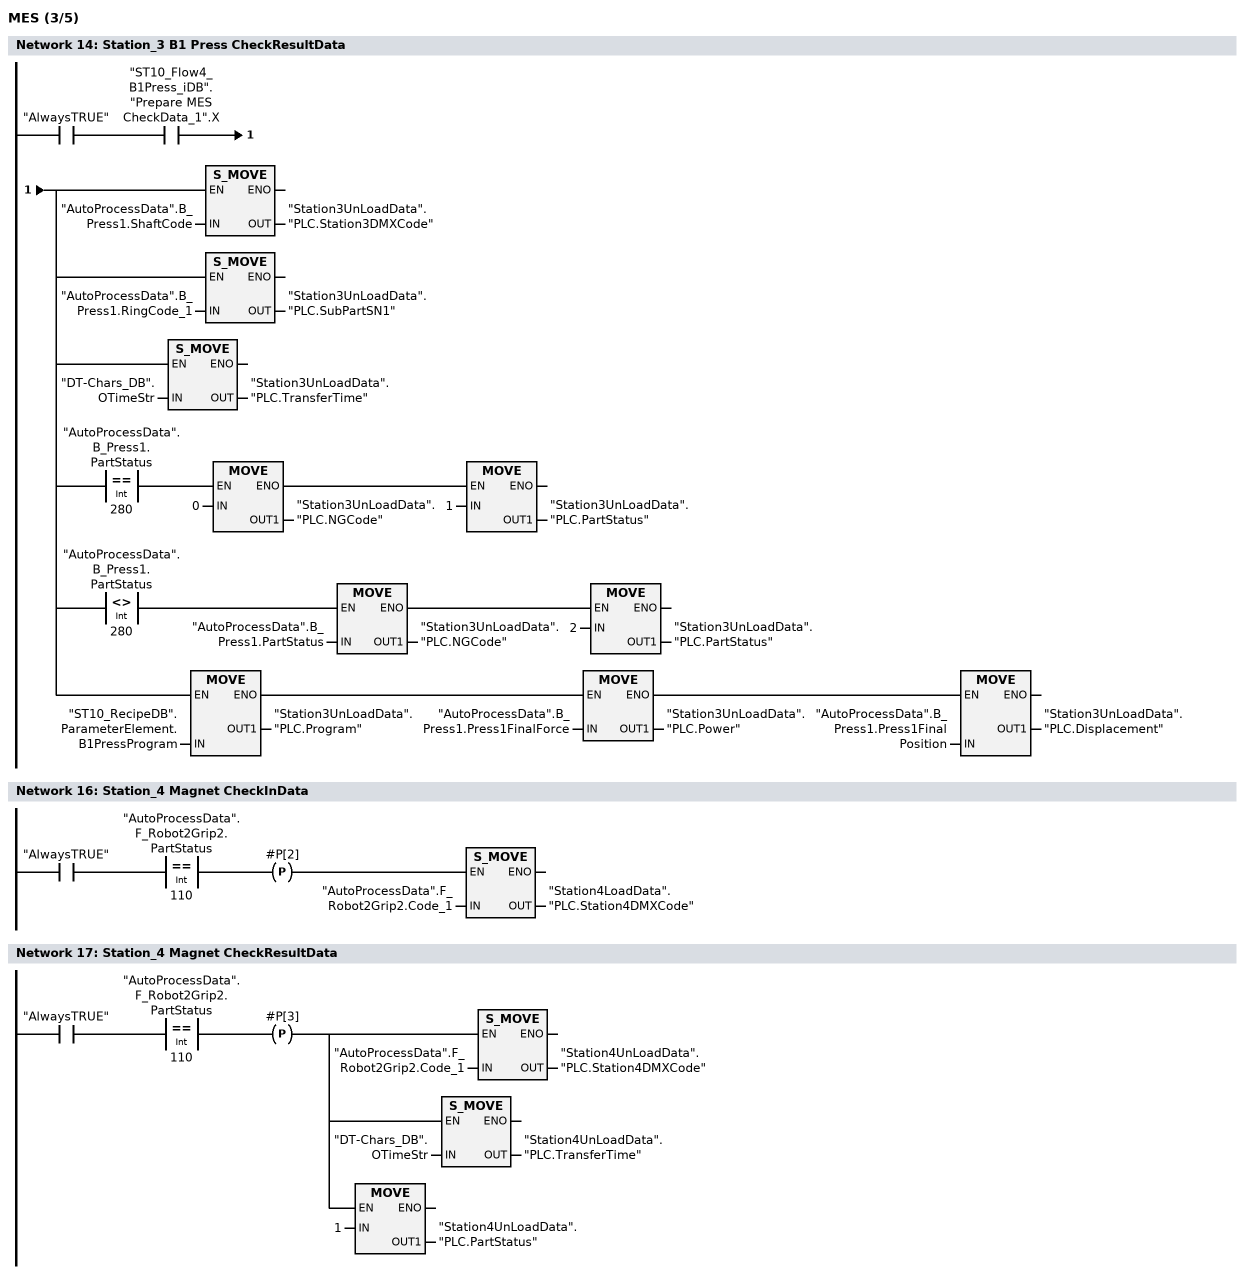
   RUNG wire#powerrail
      Contact( "AlwaysTRUE" )
      Contact( "ST10_Flow4_B1Press_iDB"."Prepare MES CheckData_1".X )
      wire#w1
      S_Move(in := "AutoProcessData".B_Press1.ShaftCode, out => "Station3UnLoadData"."PLC.Station3DMXCode")
   END_RUNG
   RUNG wire#w1
      S_Move(in := "AutoProcessData".B_Press1.RingCode_1, out => "Station3UnLoadData"."PLC.SubPartSN1")
   END_RUNG
   RUNG wire#w1
      S_Move(in := "DT-Chars_DB".OTimeStr, out => "Station3UnLoadData"."PLC.TransferTime")
   END_RUNG
   RUNG wire#w1
      { S7_Templates := "SrcType := Int" } EQ_Contact(in1 := "AutoProcessData".B_Press1.PartStatus, in2 := 280)
      Move(in := 0, out1 => "Station3UnLoadData"."PLC.NGCode")
      Move(in := 1, out1 => "Station3UnLoadData"."PLC.PartStatus")
   END_RUNG
   RUNG wire#w1
      { S7_Templates := "SrcType := Int" } NE_Contact(in1 := "AutoProcessData".B_Press1.PartStatus, in2 := 280)
      Move(in := "AutoProcessData".B_Press1.PartStatus, out1 => "Station3UnLoadData"."PLC.NGCode")
      Move(in := 2, out1 => "Station3UnLoadData"."PLC.PartStatus")
   END_RUNG
   RUNG wire#w1
      Move(in := "ST10_RecipeDB".ParameterElement.B1PressProgram, out1 => "Station3UnLoadData"."PLC.Program")
      Move(in := "AutoProcessData".B_Press1.Press1FinalForce, out1 => "Station3UnLoadData"."PLC.Power")
      Move(in := "AutoProcessData".B_Press1.Press1FinalPosition, out1 => "Station3UnLoadData"."PLC.Displacement")
   END_RUNG
   // the same network as SCL:
   #_w1 := "AlwaysTRUE" AND "ST10_Flow4_B1Press_iDB"."Prepare MES CheckData_1".X;
   IF #_w1 THEN
       "Station3UnLoadData"."PLC.Station3DMXCode" := "AutoProcessData".B_Press1.ShaftCode;
       "Station3UnLoadData"."PLC.SubPartSN1" := "AutoProcessData".B_Press1.RingCode_1;
       "Station3UnLoadData"."PLC.TransferTime" := "DT-Chars_DB".OTimeStr;
   END_IF;
   IF #_w1 AND ("AutoProcessData".B_Press1.PartStatus = 280) THEN
       "Station3UnLoadData"."PLC.NGCode" := 0;
       "Station3UnLoadData"."PLC.PartStatus" := 1;
   END_IF;
   IF #_w1 AND ("AutoProcessData".B_Press1.PartStatus <> 280) THEN
       "Station3UnLoadData"."PLC.NGCode" := "AutoProcessData".B_Press1.PartStatus;
       "Station3UnLoadData"."PLC.PartStatus" := 2;
   END_IF;
   IF #_w1 THEN
       "Station3UnLoadData"."PLC.Program" := "ST10_RecipeDB".ParameterElement.B1PressProgram;
       "Station3UnLoadData"."PLC.Power" := "AutoProcessData".B_Press1.Press1FinalForce;
       "Station3UnLoadData"."PLC.Displacement" := "AutoProcessData".B_Press1.Press1FinalPosition;
   END_IF;
END_REGION

REGION Network 16: Station_4 Magnet CheckInData
   RUNG wire#powerrail
      Contact( "AlwaysTRUE" )
      { S7_Templates := "SrcType := Int" } EQ_Contact(in1 := "AutoProcessData".F_Robot2Grip2.PartStatus, in2 := 110)
      P_Trig( #P[2] )
      S_Move(in := "AutoProcessData".F_Robot2Grip2.Code_1, out => "Station4LoadData"."PLC.Station4DMXCode")
   END_RUNG
   // the same network as SCL:
   #_w1 := "AlwaysTRUE" AND ("AutoProcessData".F_Robot2Grip2.PartStatus = 110);
   #_w2 := #_w1 AND NOT #P[2];   // rising edge
   #P[2] := #_w1;
   IF #_w2 THEN "Station4LoadData"."PLC.Station4DMXCode" := "AutoProcessData".F_Robot2Grip2.Code_1; END_IF;
END_REGION

REGION Network 17: Station_4 Magnet CheckResultData
   RUNG wire#powerrail
      Contact( "AlwaysTRUE" )
      { S7_Templates := "SrcType := Int" } EQ_Contact(in1 := "AutoProcessData".F_Robot2Grip2.PartStatus, in2 := 110)
      P_Trig( #P[3] )
      wire#w1
      S_Move(in := "AutoProcessData".F_Robot2Grip2.Code_1, out => "Station4UnLoadData"."PLC.Station4DMXCode")
   END_RUNG
   RUNG wire#w1
      S_Move(in := "DT-Chars_DB".OTimeStr, out => "Station4UnLoadData"."PLC.TransferTime")
   END_RUNG
   RUNG wire#w1
      Move(in := 1, out1 => "Station4UnLoadData"."PLC.PartStatus")
   END_RUNG
   // the same network as SCL:
   #_w1 := "AlwaysTRUE" AND ("AutoProcessData".F_Robot2Grip2.PartStatus = 110);
   #_w2 := #_w1 AND NOT #P[3];   // rising edge
   #P[3] := #_w1;
   IF #_w2 THEN
       "Station4UnLoadData"."PLC.Station4DMXCode" := "AutoProcessData".F_Robot2Grip2.Code_1;
       "Station4UnLoadData"."PLC.TransferTime" := "DT-Chars_DB".OTimeStr;
       "Station4UnLoadData"."PLC.PartStatus" := 1;
   END_IF;
END_REGION

REGION Network 19: Station_5 Glue CheckInData
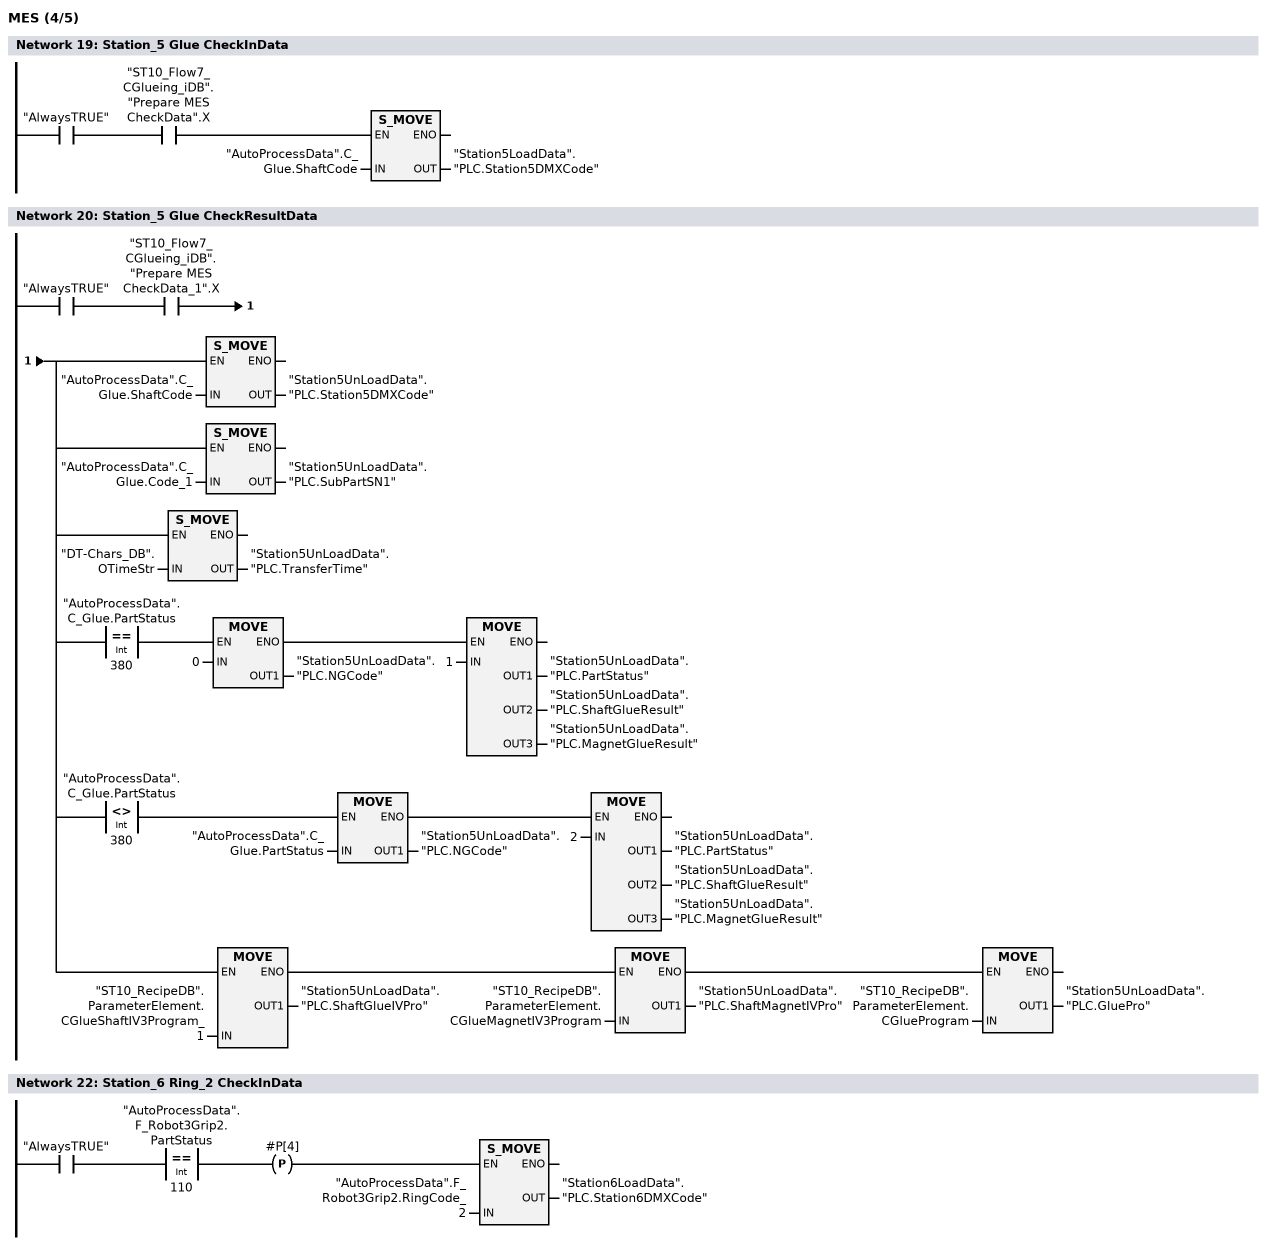
   RUNG wire#powerrail
      Contact( "AlwaysTRUE" )
      Contact( "ST10_Flow7_CGlueing_iDB"."Prepare MES CheckData".X )
      S_Move(in := "AutoProcessData".C_Glue.ShaftCode, out => "Station5LoadData"."PLC.Station5DMXCode")
   END_RUNG
   // the same network as SCL:
   IF "AlwaysTRUE" AND "ST10_Flow7_CGlueing_iDB"."Prepare MES CheckData".X THEN
       "Station5LoadData"."PLC.Station5DMXCode" := "AutoProcessData".C_Glue.ShaftCode;
   END_IF;
END_REGION

REGION Network 20: Station_5 Glue CheckResultData
   RUNG wire#powerrail
      Contact( "AlwaysTRUE" )
      Contact( "ST10_Flow7_CGlueing_iDB"."Prepare MES CheckData_1".X )
      wire#w1
      S_Move(in := "AutoProcessData".C_Glue.ShaftCode, out => "Station5UnLoadData"."PLC.Station5DMXCode")
   END_RUNG
   RUNG wire#w1
      S_Move(in := "AutoProcessData".C_Glue.Code_1, out => "Station5UnLoadData"."PLC.SubPartSN1")
   END_RUNG
   RUNG wire#w1
      S_Move(in := "DT-Chars_DB".OTimeStr, out => "Station5UnLoadData"."PLC.TransferTime")
   END_RUNG
   RUNG wire#w1
      { S7_Templates := "SrcType := Int" } EQ_Contact(in1 := "AutoProcessData".C_Glue.PartStatus, in2 := 380)
      Move(in := 0, out1 => "Station5UnLoadData"."PLC.NGCode")
      Move(in := 1, out1 => "Station5UnLoadData"."PLC.PartStatus", out2 => "Station5UnLoadData"."PLC.ShaftGlueResult", out3 => "Station5UnLoadData"."PLC.MagnetGlueResult")
   END_RUNG
   RUNG wire#w1
      { S7_Templates := "SrcType := Int" } NE_Contact(in1 := "AutoProcessData".C_Glue.PartStatus, in2 := 380)
      Move(in := "AutoProcessData".C_Glue.PartStatus, out1 => "Station5UnLoadData"."PLC.NGCode")
      Move(in := 2, out1 => "Station5UnLoadData"."PLC.PartStatus", out2 => "Station5UnLoadData"."PLC.ShaftGlueResult", out3 => "Station5UnLoadData"."PLC.MagnetGlueResult")
   END_RUNG
   RUNG wire#w1
      Move(in := "ST10_RecipeDB".ParameterElement.CGlueShaftIV3Program_1, out1 => "Station5UnLoadData"."PLC.ShaftGlueIVPro")
      Move(in := "ST10_RecipeDB".ParameterElement.CGlueMagnetIV3Program, out1 => "Station5UnLoadData"."PLC.ShaftMagnetIVPro")
      Move(in := "ST10_RecipeDB".ParameterElement.CGlueProgram, out1 => "Station5UnLoadData"."PLC.GluePro")
   END_RUNG
   // the same network as SCL:
   #_w1 := "AlwaysTRUE" AND "ST10_Flow7_CGlueing_iDB"."Prepare MES CheckData_1".X;
   IF #_w1 THEN
       "Station5UnLoadData"."PLC.Station5DMXCode" := "AutoProcessData".C_Glue.ShaftCode;
       "Station5UnLoadData"."PLC.SubPartSN1" := "AutoProcessData".C_Glue.Code_1;
       "Station5UnLoadData"."PLC.TransferTime" := "DT-Chars_DB".OTimeStr;
   END_IF;
   IF #_w1 AND ("AutoProcessData".C_Glue.PartStatus = 380) THEN
       "Station5UnLoadData"."PLC.NGCode" := 0;
       "Station5UnLoadData"."PLC.PartStatus" := 1;
       "Station5UnLoadData"."PLC.ShaftGlueResult" := 1;
       "Station5UnLoadData"."PLC.MagnetGlueResult" := 1;
   END_IF;
   IF #_w1 AND ("AutoProcessData".C_Glue.PartStatus <> 380) THEN
       "Station5UnLoadData"."PLC.NGCode" := "AutoProcessData".C_Glue.PartStatus;
       "Station5UnLoadData"."PLC.PartStatus" := 2;
       "Station5UnLoadData"."PLC.ShaftGlueResult" := 2;
       "Station5UnLoadData"."PLC.MagnetGlueResult" := 2;
   END_IF;
   IF #_w1 THEN
       "Station5UnLoadData"."PLC.ShaftGlueIVPro" := "ST10_RecipeDB".ParameterElement.CGlueShaftIV3Program_1;
       "Station5UnLoadData"."PLC.ShaftMagnetIVPro" := "ST10_RecipeDB".ParameterElement.CGlueMagnetIV3Program;
       "Station5UnLoadData"."PLC.GluePro" := "ST10_RecipeDB".ParameterElement.CGlueProgram;
   END_IF;
END_REGION

REGION Network 22: Station_6 Ring_2 CheckInData
   RUNG wire#powerrail
      Contact( "AlwaysTRUE" )
      { S7_Templates := "SrcType := Int" } EQ_Contact(in1 := "AutoProcessData".F_Robot3Grip2.PartStatus, in2 := 110)
      P_Trig( #P[4] )
      S_Move(in := "AutoProcessData".F_Robot3Grip2.RingCode_2, out => "Station6LoadData"."PLC.Station6DMXCode")
   END_RUNG
   // the same network as SCL:
   #_w1 := "AlwaysTRUE" AND ("AutoProcessData".F_Robot3Grip2.PartStatus = 110);
   #_w2 := #_w1 AND NOT #P[4];   // rising edge
   #P[4] := #_w1;
   IF #_w2 THEN
       "Station6LoadData"."PLC.Station6DMXCode" := "AutoProcessData".F_Robot3Grip2.RingCode_2;
   END_IF;
END_REGION

REGION Network 23: Station_6 Ring_2 CheckResultData
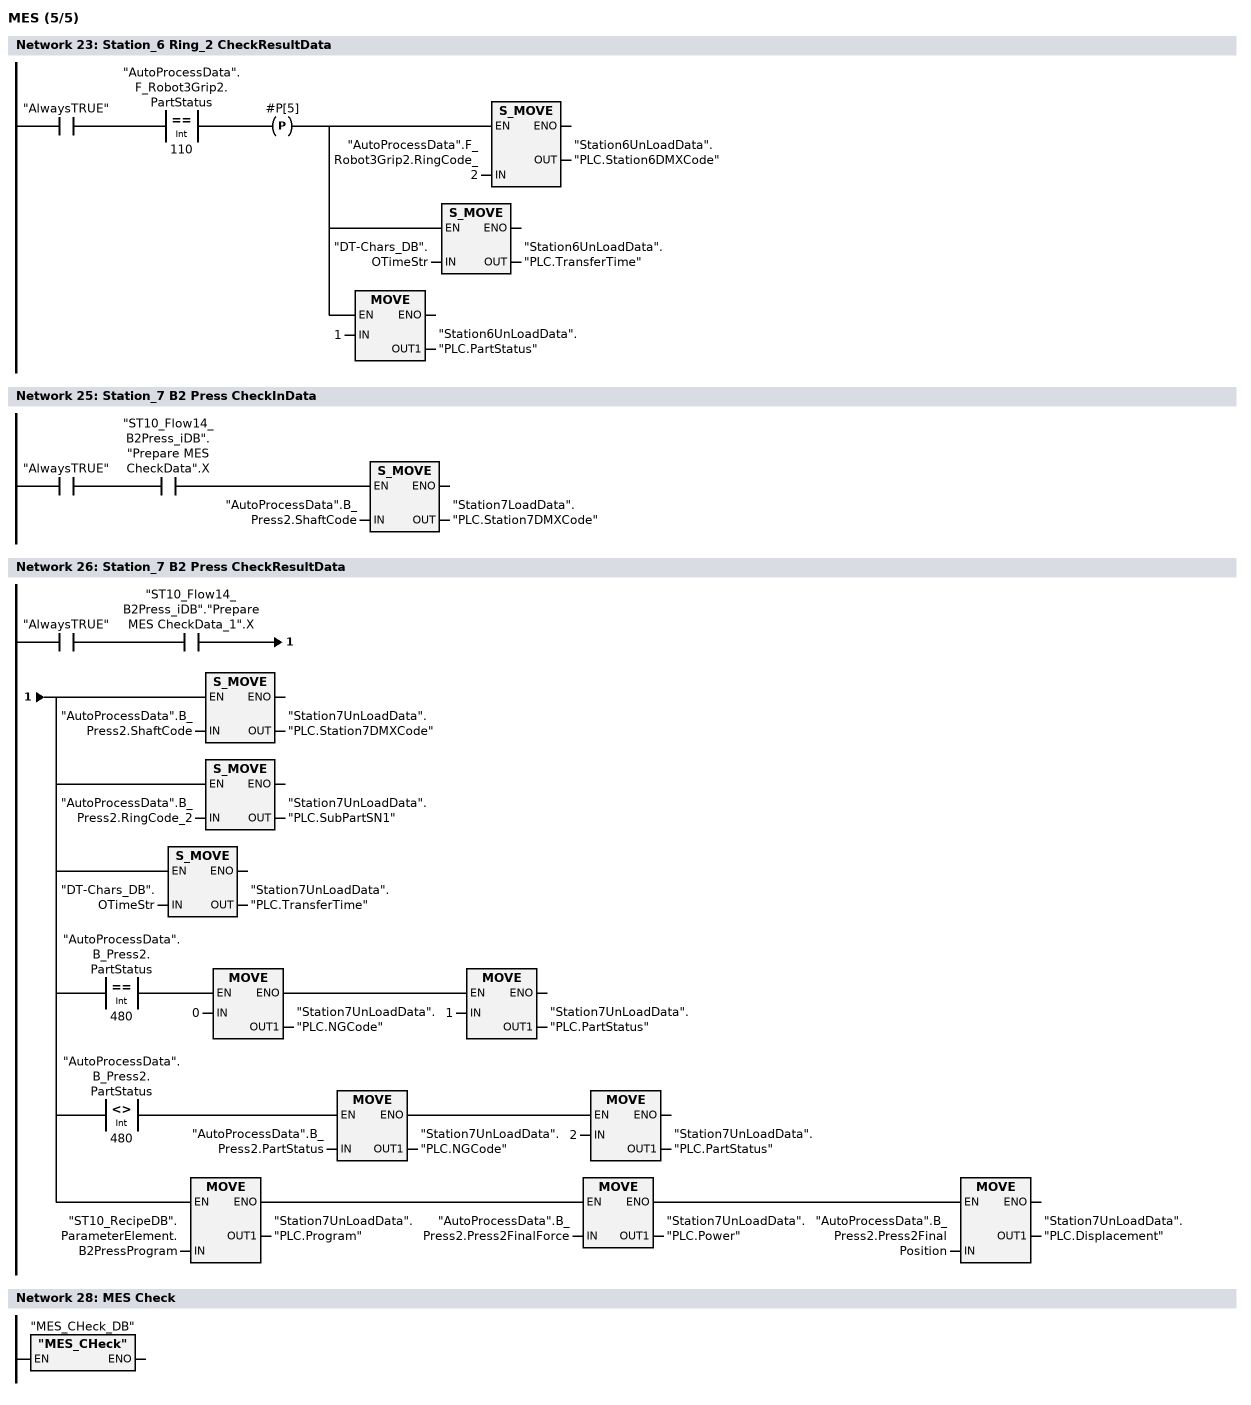
   RUNG wire#powerrail
      Contact( "AlwaysTRUE" )
      { S7_Templates := "SrcType := Int" } EQ_Contact(in1 := "AutoProcessData".F_Robot3Grip2.PartStatus, in2 := 110)
      P_Trig( #P[5] )
      wire#w1
      S_Move(in := "AutoProcessData".F_Robot3Grip2.RingCode_2, out => "Station6UnLoadData"."PLC.Station6DMXCode")
   END_RUNG
   RUNG wire#w1
      S_Move(in := "DT-Chars_DB".OTimeStr, out => "Station6UnLoadData"."PLC.TransferTime")
   END_RUNG
   RUNG wire#w1
      Move(in := 1, out1 => "Station6UnLoadData"."PLC.PartStatus")
   END_RUNG
   // the same network as SCL:
   #_w1 := "AlwaysTRUE" AND ("AutoProcessData".F_Robot3Grip2.PartStatus = 110);
   #_w2 := #_w1 AND NOT #P[5];   // rising edge
   #P[5] := #_w1;
   IF #_w2 THEN
       "Station6UnLoadData"."PLC.Station6DMXCode" := "AutoProcessData".F_Robot3Grip2.RingCode_2;
       "Station6UnLoadData"."PLC.TransferTime" := "DT-Chars_DB".OTimeStr;
       "Station6UnLoadData"."PLC.PartStatus" := 1;
   END_IF;
END_REGION

REGION Network 25: Station_7 B2 Press CheckInData
   RUNG wire#powerrail
      Contact( "AlwaysTRUE" )
      Contact( "ST10_Flow14_B2Press_iDB"."Prepare MES CheckData".X )
      S_Move(in := "AutoProcessData".B_Press2.ShaftCode, out => "Station7LoadData"."PLC.Station7DMXCode")
   END_RUNG
   // the same network as SCL:
   IF "AlwaysTRUE" AND "ST10_Flow14_B2Press_iDB"."Prepare MES CheckData".X THEN
       "Station7LoadData"."PLC.Station7DMXCode" := "AutoProcessData".B_Press2.ShaftCode;
   END_IF;
END_REGION

REGION Network 26: Station_7 B2 Press CheckResultData
   RUNG wire#powerrail
      Contact( "AlwaysTRUE" )
      Contact( "ST10_Flow14_B2Press_iDB"."Prepare MES CheckData_1".X )
      wire#w1
      S_Move(in := "AutoProcessData".B_Press2.ShaftCode, out => "Station7UnLoadData"."PLC.Station7DMXCode")
   END_RUNG
   RUNG wire#w1
      S_Move(in := "AutoProcessData".B_Press2.RingCode_2, out => "Station7UnLoadData"."PLC.SubPartSN1")
   END_RUNG
   RUNG wire#w1
      S_Move(in := "DT-Chars_DB".OTimeStr, out => "Station7UnLoadData"."PLC.TransferTime")
   END_RUNG
   RUNG wire#w1
      { S7_Templates := "SrcType := Int" } EQ_Contact(in1 := "AutoProcessData".B_Press2.PartStatus, in2 := 480)
      Move(in := 0, out1 => "Station7UnLoadData"."PLC.NGCode")
      Move(in := 1, out1 => "Station7UnLoadData"."PLC.PartStatus")
   END_RUNG
   RUNG wire#w1
      { S7_Templates := "SrcType := Int" } NE_Contact(in1 := "AutoProcessData".B_Press2.PartStatus, in2 := 480)
      Move(in := "AutoProcessData".B_Press2.PartStatus, out1 => "Station7UnLoadData"."PLC.NGCode")
      Move(in := 2, out1 => "Station7UnLoadData"."PLC.PartStatus")
   END_RUNG
   RUNG wire#w1
      Move(in := "ST10_RecipeDB".ParameterElement.B2PressProgram, out1 => "Station7UnLoadData"."PLC.Program")
      Move(in := "AutoProcessData".B_Press2.Press2FinalForce, out1 => "Station7UnLoadData"."PLC.Power")
      Move(in := "AutoProcessData".B_Press2.Press2FinalPosition, out1 => "Station7UnLoadData"."PLC.Displacement")
   END_RUNG
   // the same network as SCL:
   #_w1 := "AlwaysTRUE" AND "ST10_Flow14_B2Press_iDB"."Prepare MES CheckData_1".X;
   IF #_w1 THEN
       "Station7UnLoadData"."PLC.Station7DMXCode" := "AutoProcessData".B_Press2.ShaftCode;
       "Station7UnLoadData"."PLC.SubPartSN1" := "AutoProcessData".B_Press2.RingCode_2;
       "Station7UnLoadData"."PLC.TransferTime" := "DT-Chars_DB".OTimeStr;
   END_IF;
   IF #_w1 AND ("AutoProcessData".B_Press2.PartStatus = 480) THEN
       "Station7UnLoadData"."PLC.NGCode" := 0;
       "Station7UnLoadData"."PLC.PartStatus" := 1;
   END_IF;
   IF #_w1 AND ("AutoProcessData".B_Press2.PartStatus <> 480) THEN
       "Station7UnLoadData"."PLC.NGCode" := "AutoProcessData".B_Press2.PartStatus;
       "Station7UnLoadData"."PLC.PartStatus" := 2;
   END_IF;
   IF #_w1 THEN
       "Station7UnLoadData"."PLC.Program" := "ST10_RecipeDB".ParameterElement.B2PressProgram;
       "Station7UnLoadData"."PLC.Power" := "AutoProcessData".B_Press2.Press2FinalForce;
       "Station7UnLoadData"."PLC.Displacement" := "AutoProcessData".B_Press2.Press2FinalPosition;
   END_IF;
END_REGION

REGION Network 28: MES Check
   RUNG wire#powerrail
      "MES_CHeck_DB"()
   END_RUNG
   // the same network as SCL:
   "MES_CHeck_DB"();   // "MES_CHeck"
END_REGION
END_FUNCTION

FUNCTION_BLOCK "DT-Chars"   // FB2360, SCL
{ S7_Optimized_Access := 'FALSE' }
// stored: AutoNumber false, SetENOAutomatically false
   VAR_INPUT
      YEAR : Int;
      MONTH : Int;
      DAY : Int;
      HH : Int;
      MM : Int;
      SS : Int;
   END_VAR
   VAR_OUTPUT
      Year_Byte1 : Char;
      Year_Byte2 : Char;
      Month_Byte1 : Char;
      Month_Byte2 : Char;
      Days_Byte1 : Char;
      Days_Byte2 : Char;
      HH_Byte1 : Char;
      HH_Byte2 : Char;
      MM_Byte1 : Char;
      MM_Byte2 : Char;
      SS_Byte1 : Char;
      SS_Byte2 : Char;
      CalculateDays_Byte1 : Char;   // 一年中的第几天
      CalculateDays_Byte2 : Char;   // 一年中的第几天
      CalculateDays_Byte3 : Char;   // 一年中的第几天
      Error_Code : Int;
      Year_Byte3 : String[1];
      Year_Byte4 : String[1];
      Month_Byte3 : String[1];
      Month_Byte4 : String[1];
      Days_Byte3 : String[1];
      Days_Byte4 : String[1];
      HH_Byte3 : String[1];
      HH_Byte4 : String[1];
      MM_Byte3 : String[1];
      MM_Byte4 : String[1];
      SS_Byte3 : String[1];
      SS_Byte4 : String[1];
      CalculateDays_Byte4 : String[1];
      CalculateDays_Byte5 : String[1];
      CalculateDays_Byte6 : String[1];
      OTimeStr : String[20];
   END_VAR
   VAR
      Sum_Days : Int;
      Sum_Year : Int;
   END_VAR
   VAR_TEMP
      Input_1_BCD : Word;
      Input_2_BCD : Word;
      Input_3_BCD : Word;
      Input_4_BCD : Word;
      Input_5_BCD : Word;
      Input_6_BCD : Word;
      Input_7_BCD : Word;
   END_VAR
BEGIN
   #Input_1_BCD := INT_TO_BCD16(#YEAR);
   #Year_Byte2 := INT_TO_BYTE(#YEAR MOD 10 + 48);
   #Year_Byte1 := INT_TO_BYTE(WORD_TO_INT(SHR(IN := #Input_1_BCD, N := 4)) + 48);


   #Input_2_BCD := INT_TO_BCD16(#MONTH);
   #Month_Byte2 := INT_TO_BYTE(#MONTH MOD 10 + 48);
   #Month_Byte1 := INT_TO_BYTE(WORD_TO_INT(SHR(IN := #Input_2_BCD, N := 4)) + 48);

   #Input_3_BCD := INT_TO_BCD16(#DAY);
   #Days_Byte2 := INT_TO_BYTE(#DAY MOD 10 + 48);
   #Days_Byte1 := INT_TO_BYTE(WORD_TO_INT(SHR(IN := #Input_3_BCD, N := 4)) + 48);

   #Input_4_BCD := INT_TO_BCD16(#HH);
   #HH_Byte2 := INT_TO_BYTE(#HH MOD 10 + 48);
   #HH_Byte1 := INT_TO_BYTE(WORD_TO_INT(SHR(IN := #Input_4_BCD, N := 4)) + 48);

   #Input_5_BCD := INT_TO_BCD16(#MM);
   #MM_Byte2 := INT_TO_BYTE(#MM MOD 10 + 48);
   #MM_Byte1 := INT_TO_BYTE(WORD_TO_INT(SHR(IN := #Input_5_BCD, N := 4)) + 48);

   #Input_6_BCD := INT_TO_BCD16(#SS);
   #SS_Byte2 := INT_TO_BYTE(#SS MOD 10 + 48);
   #SS_Byte1 := INT_TO_BYTE(WORD_TO_INT(SHR(IN := #Input_6_BCD, N := 4)) + 48);

   #Sum_Days := 0;//初始值
   #Sum_Year := 2000 + #YEAR;
   CASE #MONTH OF
       12:
           #Sum_Days := 31 + 28 + 31 + 30 + 31 + 30 + 31 + 31 + 30 + 31 + 30 + #DAY;
       11:
           #Sum_Days := 31 + 28 + 31 + 30 + 31 + 30 + 31 + 31 + 30 + 31 + #DAY;
       10:
           #Sum_Days := 31 + 28 + 31 + 30 + 31 + 30 + 31 + 31 + 30 + #DAY;
       9:
           #Sum_Days := 31 + 28 + 31 + 30 + 31 + 30 + 31 + 31 + #DAY;
       8:
           #Sum_Days := 31 + 28 + 31 + 30 + 31 + 30 + 31 + #DAY;
       7:
           #Sum_Days := 31 + 28 + 31 + 30 + 31 + 30 + #DAY;
       6:
           #Sum_Days := 31 + 28 + 31 + 30 + 31 + #DAY;
       5:
           #Sum_Days := 31 + 28 + 31 + 30 + #DAY;
       4:
           #Sum_Days := 31 + 28 + 31 + #DAY;
       3:
           #Sum_Days := 31 + 28 + #DAY;
       2:
           #Sum_Days := 31 + #DAY;
       1:
           #Sum_Days := #DAY;

   END_CASE;

   //判断是否是闰年 闰年2月29天
   IF (#Sum_Year MOD 4=0)AND(#Sum_Year MOD 100<>0)OR(#Sum_Year MOD 400=0)AND(#MONTH > 2) THEN
           // Statement section IF 
       #Sum_Days := #Sum_Days +1;//闰年2月+1    
   END_IF;

   #Input_4_BCD:=INT_TO_BCD16(#Sum_Days);
   #CalculateDays_Byte3 := INT_TO_BYTE(WORD_TO_INT(SHR(IN := (#Input_4_BCD AND 16#000F), N :=0 )) + 48);
   #CalculateDays_Byte2 := INT_TO_BYTE(WORD_TO_INT(SHR(IN := (#Input_4_BCD AND 16#00F0), N := 4)) + 48);
   #CalculateDays_Byte1 := INT_TO_BYTE(WORD_TO_INT(SHR(IN := (#Input_4_BCD AND 16#0F00), N := 8)) + 48);

   #Year_Byte3 := CHAR_TO_STRING(#Year_Byte1);
   #Year_Byte4 := CHAR_TO_STRING(#Year_Byte2);

   #Month_Byte3 := CHAR_TO_STRING(#Month_Byte1);
   #Month_Byte4 := CHAR_TO_STRING(#Month_Byte2);

   #Days_Byte3 := CHAR_TO_STRING(#Days_Byte1);
   #Days_Byte4 := CHAR_TO_STRING(#Days_Byte2);

   #HH_Byte3 := CHAR_TO_STRING(#HH_Byte1);
   #HH_Byte4 := CHAR_TO_STRING(#HH_Byte2);

   #MM_Byte3 := CHAR_TO_STRING(#MM_Byte1);
   #MM_Byte4 := CHAR_TO_STRING(#MM_Byte2);

   #SS_Byte3 := CHAR_TO_STRING(#SS_Byte1);
   #SS_Byte4 := CHAR_TO_STRING(#SS_Byte2);

   #CalculateDays_Byte4 := CHAR_TO_STRING(#CalculateDays_Byte1);
   #CalculateDays_Byte5 := CHAR_TO_STRING(#CalculateDays_Byte2);
   #CalculateDays_Byte6 := CHAR_TO_STRING(#CalculateDays_Byte3);


   #OTimeStr := CONCAT(IN1 := '20', IN2 := #Year_Byte3, IN3 := #Year_Byte4, IN4 := '-',
                                    IN5 := #Month_Byte3, IN6 := #Month_Byte4, IN7 := '-',
                                    IN8 := #Days_Byte3, IN9 := #Days_Byte4, IN10 := ' ',
                                    IN11 := #HH_Byte3, IN12 := #HH_Byte4, IN13 := ':',
                                    IN14 := #MM_Byte3, IN15 := #MM_Byte4, IN16 := ':',
                                    IN17 := #SS_Byte3, IN18 := #SS_Byte4);
END_FUNCTION_BLOCK

FUNCTION_BLOCK "MES_CHeck"   // FB111, LAD
{ S7_Optimized_Access := 'TRUE' }
VERSION : 0.1
// stored: AutoNumber false, IsIECCheckEnabled false, IsRetainMemResEnabled false, MemoryReserve 100, SetENOAutomatically false, UDAEnableTagReadback false
   VAR
      Station_1 : "MES Check_fb";   // *
      Station_2 : "MES Check_fb";   // *
      Station_3 : "MES Check_fb";   // *
      Station_4 : "MES Check_fb";   // *
      Station_5 : "MES Check_fb";   // *
      Station_6 : "MES Check_fb";   // *
      Station_7 : "MES Check_fb";   // *
      Station_8 : "MES Check_fb";   // *
   END_VAR
BEGIN

REGION Network 1: Station_1 shaft_1
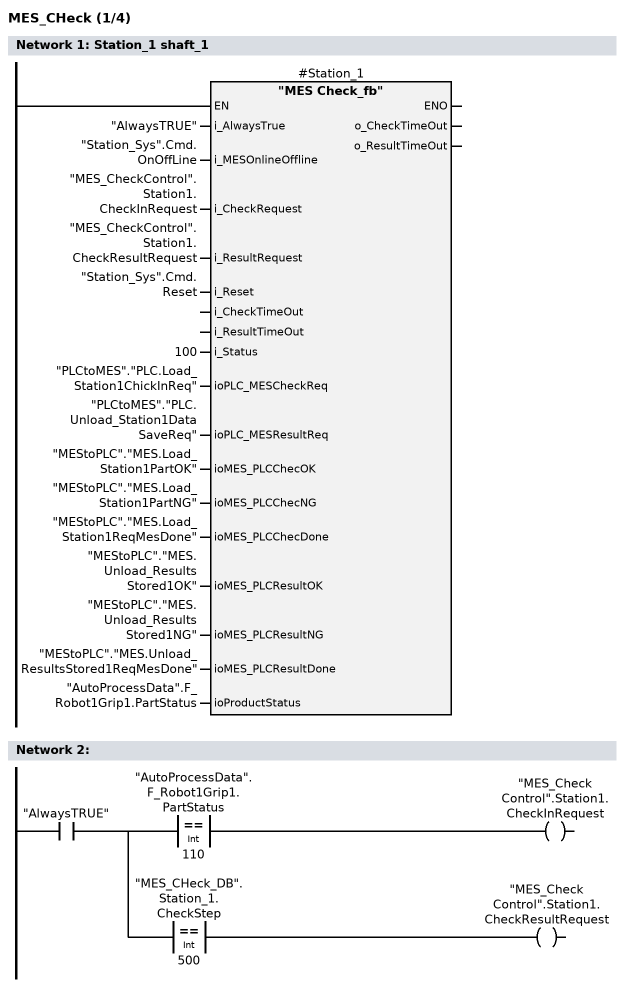
   RUNG wire#powerrail
      #Station_1(i_AlwaysTrue := "AlwaysTRUE", i_MESOnlineOffline := "Station_Sys".Cmd.OnOffLine, i_CheckRequest := "MES_CheckControl".Station1.CheckInRequest, i_ResultRequest := "MES_CheckControl".Station1.CheckResultRequest, i_Reset := "Station_Sys".Cmd.Reset, i_CheckTimeOut :=, i_ResultTimeOut :=, i_Status := 100, ioPLC_MESCheckReq := "PLCtoMES"."PLC.Load_Station1ChickInReq", ioPLC_MESResultReq := "PLCtoMES"."PLC.Unload_Station1DataSaveReq", ioMES_PLCChecOK := "MEStoPLC"."MES.Load_Station1PartOK", ioMES_PLCChecNG := "MEStoPLC"."MES.Load_Station1PartNG", ioMES_PLCChecDone := "MEStoPLC"."MES.Load_Station1ReqMesDone", ioMES_PLCResultOK := "MEStoPLC"."MES.Unload_ResultsStored1OK", ioMES_PLCResultNG := "MEStoPLC"."MES.Unload_ResultsStored1NG", ioMES_PLCResultDone := "MEStoPLC"."MES.Unload_ResultsStored1ReqMesDone", ioProductStatus := "AutoProcessData".F_Robot1Grip1.PartStatus, o_CheckTimeOut =>, o_ResultTimeOut =>)
   END_RUNG
   // the same network as SCL:
   #Station_1(i_AlwaysTrue := "AlwaysTRUE",   // "MES Check_fb"
              i_MESOnlineOffline := "Station_Sys".Cmd.OnOffLine,
              i_CheckRequest := "MES_CheckControl".Station1.CheckInRequest,
              i_ResultRequest := "MES_CheckControl".Station1.CheckResultRequest,
              i_Reset := "Station_Sys".Cmd.Reset,
              i_Status := 100,
              ioPLC_MESCheckReq := "PLCtoMES"."PLC.Load_Station1ChickInReq",
              ioPLC_MESResultReq := "PLCtoMES"."PLC.Unload_Station1DataSaveReq",
              ioMES_PLCChecOK := "MEStoPLC"."MES.Load_Station1PartOK",
              ioMES_PLCChecNG := "MEStoPLC"."MES.Load_Station1PartNG",
              ioMES_PLCChecDone := "MEStoPLC"."MES.Load_Station1ReqMesDone",
              ioMES_PLCResultOK := "MEStoPLC"."MES.Unload_ResultsStored1OK",
              ioMES_PLCResultNG := "MEStoPLC"."MES.Unload_ResultsStored1NG",
              ioMES_PLCResultDone := "MEStoPLC"."MES.Unload_ResultsStored1ReqMesDone",
              ioProductStatus := "AutoProcessData".F_Robot1Grip1.PartStatus);
END_REGION

REGION Network 2
   RUNG wire#powerrail
      Contact( "AlwaysTRUE" )
      wire#w1
      { S7_Templates := "SrcType := Int" } EQ_Contact(in1 := "AutoProcessData".F_Robot1Grip1.PartStatus, in2 := 110)
      Coil( "MES_CheckControl".Station1.CheckInRequest )
   END_RUNG
   RUNG wire#w1
      { S7_Templates := "SrcType := Int" } EQ_Contact(in1 := "MES_CHeck_DB".Station_1.CheckStep, in2 := 500)
      Coil( "MES_CheckControl".Station1.CheckResultRequest )
   END_RUNG
   // the same network as SCL:
   "MES_CheckControl".Station1.CheckInRequest := "AlwaysTRUE" AND ("AutoProcessData".F_Robot1Grip1.PartStatus = 110);
   "MES_CheckControl".Station1.CheckResultRequest := "AlwaysTRUE" AND ("MES_CHeck_DB".Station_1.CheckStep = 500);
END_REGION

REGION Network 3: Station_2 Ring_1
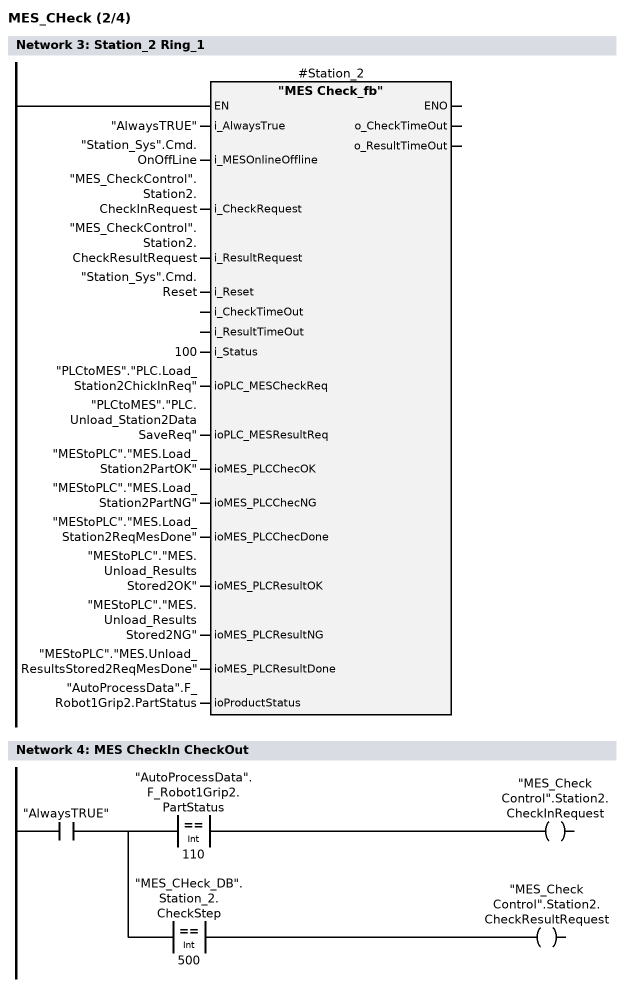
   RUNG wire#powerrail
      #Station_2(i_AlwaysTrue := "AlwaysTRUE", i_MESOnlineOffline := "Station_Sys".Cmd.OnOffLine, i_CheckRequest := "MES_CheckControl".Station2.CheckInRequest, i_ResultRequest := "MES_CheckControl".Station2.CheckResultRequest, i_Reset := "Station_Sys".Cmd.Reset, i_CheckTimeOut :=, i_ResultTimeOut :=, i_Status := 100, ioPLC_MESCheckReq := "PLCtoMES"."PLC.Load_Station2ChickInReq", ioPLC_MESResultReq := "PLCtoMES"."PLC.Unload_Station2DataSaveReq", ioMES_PLCChecOK := "MEStoPLC"."MES.Load_Station2PartOK", ioMES_PLCChecNG := "MEStoPLC"."MES.Load_Station2PartNG", ioMES_PLCChecDone := "MEStoPLC"."MES.Load_Station2ReqMesDone", ioMES_PLCResultOK := "MEStoPLC"."MES.Unload_ResultsStored2OK", ioMES_PLCResultNG := "MEStoPLC"."MES.Unload_ResultsStored2NG", ioMES_PLCResultDone := "MEStoPLC"."MES.Unload_ResultsStored2ReqMesDone", ioProductStatus := "AutoProcessData".F_Robot1Grip2.PartStatus, o_CheckTimeOut =>, o_ResultTimeOut =>)
   END_RUNG
   // the same network as SCL:
   #Station_2(i_AlwaysTrue := "AlwaysTRUE",   // "MES Check_fb"
              i_MESOnlineOffline := "Station_Sys".Cmd.OnOffLine,
              i_CheckRequest := "MES_CheckControl".Station2.CheckInRequest,
              i_ResultRequest := "MES_CheckControl".Station2.CheckResultRequest,
              i_Reset := "Station_Sys".Cmd.Reset,
              i_Status := 100,
              ioPLC_MESCheckReq := "PLCtoMES"."PLC.Load_Station2ChickInReq",
              ioPLC_MESResultReq := "PLCtoMES"."PLC.Unload_Station2DataSaveReq",
              ioMES_PLCChecOK := "MEStoPLC"."MES.Load_Station2PartOK",
              ioMES_PLCChecNG := "MEStoPLC"."MES.Load_Station2PartNG",
              ioMES_PLCChecDone := "MEStoPLC"."MES.Load_Station2ReqMesDone",
              ioMES_PLCResultOK := "MEStoPLC"."MES.Unload_ResultsStored2OK",
              ioMES_PLCResultNG := "MEStoPLC"."MES.Unload_ResultsStored2NG",
              ioMES_PLCResultDone := "MEStoPLC"."MES.Unload_ResultsStored2ReqMesDone",
              ioProductStatus := "AutoProcessData".F_Robot1Grip2.PartStatus);
END_REGION

REGION Network 4: MES CheckIn CheckOut
   RUNG wire#powerrail
      Contact( "AlwaysTRUE" )
      wire#w1
      { S7_Templates := "SrcType := Int" } EQ_Contact(in1 := "AutoProcessData".F_Robot1Grip2.PartStatus, in2 := 110)
      Coil( "MES_CheckControl".Station2.CheckInRequest )
   END_RUNG
   RUNG wire#w1
      { S7_Templates := "SrcType := Int" } EQ_Contact(in1 := "MES_CHeck_DB".Station_2.CheckStep, in2 := 500)
      Coil( "MES_CheckControl".Station2.CheckResultRequest )
   END_RUNG
   // the same network as SCL:
   "MES_CheckControl".Station2.CheckInRequest := "AlwaysTRUE" AND ("AutoProcessData".F_Robot1Grip2.PartStatus = 110);
   "MES_CheckControl".Station2.CheckResultRequest := "AlwaysTRUE" AND ("MES_CHeck_DB".Station_2.CheckStep = 500);
END_REGION

REGION Network 5: Station_4 Magnet
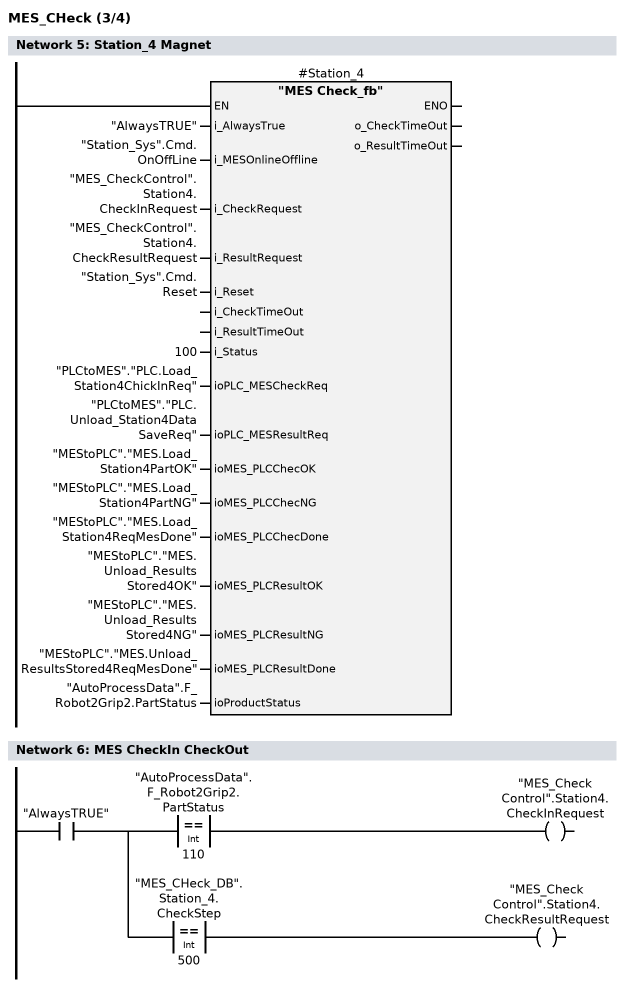
   RUNG wire#powerrail
      #Station_4(i_AlwaysTrue := "AlwaysTRUE", i_MESOnlineOffline := "Station_Sys".Cmd.OnOffLine, i_CheckRequest := "MES_CheckControl".Station4.CheckInRequest, i_ResultRequest := "MES_CheckControl".Station4.CheckResultRequest, i_Reset := "Station_Sys".Cmd.Reset, i_CheckTimeOut :=, i_ResultTimeOut :=, i_Status := 100, ioPLC_MESCheckReq := "PLCtoMES"."PLC.Load_Station4ChickInReq", ioPLC_MESResultReq := "PLCtoMES"."PLC.Unload_Station4DataSaveReq", ioMES_PLCChecOK := "MEStoPLC"."MES.Load_Station4PartOK", ioMES_PLCChecNG := "MEStoPLC"."MES.Load_Station4PartNG", ioMES_PLCChecDone := "MEStoPLC"."MES.Load_Station4ReqMesDone", ioMES_PLCResultOK := "MEStoPLC"."MES.Unload_ResultsStored4OK", ioMES_PLCResultNG := "MEStoPLC"."MES.Unload_ResultsStored4NG", ioMES_PLCResultDone := "MEStoPLC"."MES.Unload_ResultsStored4ReqMesDone", ioProductStatus := "AutoProcessData".F_Robot2Grip2.PartStatus, o_CheckTimeOut =>, o_ResultTimeOut =>)
   END_RUNG
   // the same network as SCL:
   #Station_4(i_AlwaysTrue := "AlwaysTRUE",   // "MES Check_fb"
              i_MESOnlineOffline := "Station_Sys".Cmd.OnOffLine,
              i_CheckRequest := "MES_CheckControl".Station4.CheckInRequest,
              i_ResultRequest := "MES_CheckControl".Station4.CheckResultRequest,
              i_Reset := "Station_Sys".Cmd.Reset,
              i_Status := 100,
              ioPLC_MESCheckReq := "PLCtoMES"."PLC.Load_Station4ChickInReq",
              ioPLC_MESResultReq := "PLCtoMES"."PLC.Unload_Station4DataSaveReq",
              ioMES_PLCChecOK := "MEStoPLC"."MES.Load_Station4PartOK",
              ioMES_PLCChecNG := "MEStoPLC"."MES.Load_Station4PartNG",
              ioMES_PLCChecDone := "MEStoPLC"."MES.Load_Station4ReqMesDone",
              ioMES_PLCResultOK := "MEStoPLC"."MES.Unload_ResultsStored4OK",
              ioMES_PLCResultNG := "MEStoPLC"."MES.Unload_ResultsStored4NG",
              ioMES_PLCResultDone := "MEStoPLC"."MES.Unload_ResultsStored4ReqMesDone",
              ioProductStatus := "AutoProcessData".F_Robot2Grip2.PartStatus);
END_REGION

REGION Network 6: MES CheckIn CheckOut
   RUNG wire#powerrail
      Contact( "AlwaysTRUE" )
      wire#w1
      { S7_Templates := "SrcType := Int" } EQ_Contact(in1 := "AutoProcessData".F_Robot2Grip2.PartStatus, in2 := 110)
      Coil( "MES_CheckControl".Station4.CheckInRequest )
   END_RUNG
   RUNG wire#w1
      { S7_Templates := "SrcType := Int" } EQ_Contact(in1 := "MES_CHeck_DB".Station_4.CheckStep, in2 := 500)
      Coil( "MES_CheckControl".Station4.CheckResultRequest )
   END_RUNG
   // the same network as SCL:
   "MES_CheckControl".Station4.CheckInRequest := "AlwaysTRUE" AND ("AutoProcessData".F_Robot2Grip2.PartStatus = 110);
   "MES_CheckControl".Station4.CheckResultRequest := "AlwaysTRUE" AND ("MES_CHeck_DB".Station_4.CheckStep = 500);
END_REGION

REGION Network 7: Station_6 Ring_2
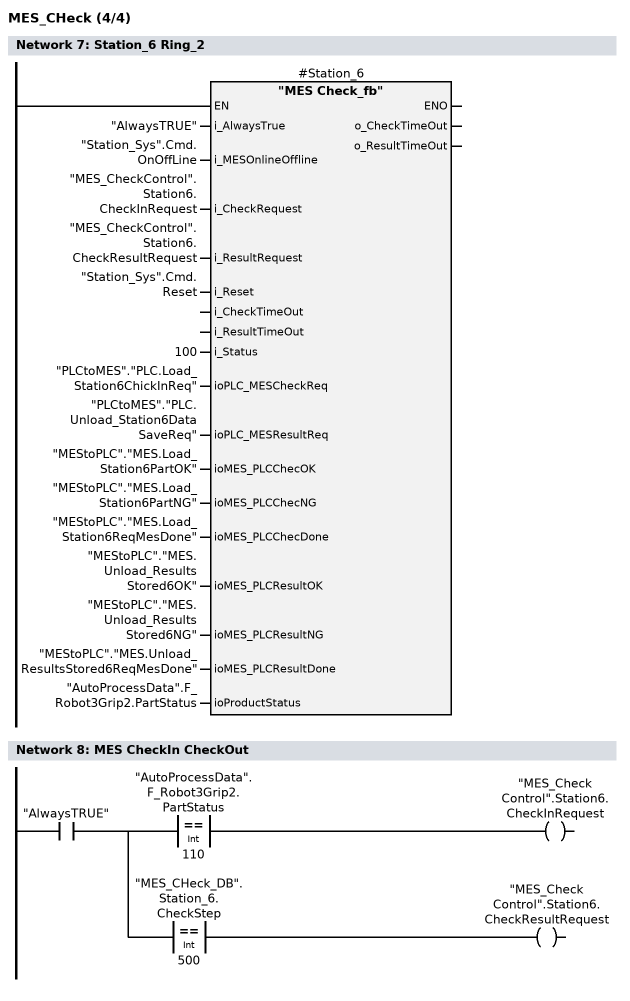
   RUNG wire#powerrail
      #Station_6(i_AlwaysTrue := "AlwaysTRUE", i_MESOnlineOffline := "Station_Sys".Cmd.OnOffLine, i_CheckRequest := "MES_CheckControl".Station6.CheckInRequest, i_ResultRequest := "MES_CheckControl".Station6.CheckResultRequest, i_Reset := "Station_Sys".Cmd.Reset, i_CheckTimeOut :=, i_ResultTimeOut :=, i_Status := 100, ioPLC_MESCheckReq := "PLCtoMES"."PLC.Load_Station6ChickInReq", ioPLC_MESResultReq := "PLCtoMES"."PLC.Unload_Station6DataSaveReq", ioMES_PLCChecOK := "MEStoPLC"."MES.Load_Station6PartOK", ioMES_PLCChecNG := "MEStoPLC"."MES.Load_Station6PartNG", ioMES_PLCChecDone := "MEStoPLC"."MES.Load_Station6ReqMesDone", ioMES_PLCResultOK := "MEStoPLC"."MES.Unload_ResultsStored6OK", ioMES_PLCResultNG := "MEStoPLC"."MES.Unload_ResultsStored6NG", ioMES_PLCResultDone := "MEStoPLC"."MES.Unload_ResultsStored6ReqMesDone", ioProductStatus := "AutoProcessData".F_Robot3Grip2.PartStatus, o_CheckTimeOut =>, o_ResultTimeOut =>)
   END_RUNG
   // the same network as SCL:
   #Station_6(i_AlwaysTrue := "AlwaysTRUE",   // "MES Check_fb"
              i_MESOnlineOffline := "Station_Sys".Cmd.OnOffLine,
              i_CheckRequest := "MES_CheckControl".Station6.CheckInRequest,
              i_ResultRequest := "MES_CheckControl".Station6.CheckResultRequest,
              i_Reset := "Station_Sys".Cmd.Reset,
              i_Status := 100,
              ioPLC_MESCheckReq := "PLCtoMES"."PLC.Load_Station6ChickInReq",
              ioPLC_MESResultReq := "PLCtoMES"."PLC.Unload_Station6DataSaveReq",
              ioMES_PLCChecOK := "MEStoPLC"."MES.Load_Station6PartOK",
              ioMES_PLCChecNG := "MEStoPLC"."MES.Load_Station6PartNG",
              ioMES_PLCChecDone := "MEStoPLC"."MES.Load_Station6ReqMesDone",
              ioMES_PLCResultOK := "MEStoPLC"."MES.Unload_ResultsStored6OK",
              ioMES_PLCResultNG := "MEStoPLC"."MES.Unload_ResultsStored6NG",
              ioMES_PLCResultDone := "MEStoPLC"."MES.Unload_ResultsStored6ReqMesDone",
              ioProductStatus := "AutoProcessData".F_Robot3Grip2.PartStatus);
END_REGION

REGION Network 8: MES CheckIn CheckOut
   RUNG wire#powerrail
      Contact( "AlwaysTRUE" )
      wire#w1
      { S7_Templates := "SrcType := Int" } EQ_Contact(in1 := "AutoProcessData".F_Robot3Grip2.PartStatus, in2 := 110)
      Coil( "MES_CheckControl".Station6.CheckInRequest )
   END_RUNG
   RUNG wire#w1
      { S7_Templates := "SrcType := Int" } EQ_Contact(in1 := "MES_CHeck_DB".Station_6.CheckStep, in2 := 500)
      Coil( "MES_CheckControl".Station6.CheckResultRequest )
   END_RUNG
   // the same network as SCL:
   "MES_CheckControl".Station6.CheckInRequest := "AlwaysTRUE" AND ("AutoProcessData".F_Robot3Grip2.PartStatus = 110);
   "MES_CheckControl".Station6.CheckResultRequest := "AlwaysTRUE" AND ("MES_CHeck_DB".Station_6.CheckStep = 500);
END_REGION
END_FUNCTION_BLOCK

FUNCTION_BLOCK "MES Check_fb"   // FB110, LAD
{ S7_Optimized_Access := 'TRUE' }
// stored: AutoNumber false, MemoryReserve 100, SetENOAutomatically false
   VAR_INPUT
      i_AlwaysTrue : Bool;
      i_MESOnlineOffline : Bool;
      i_CheckRequest : Bool;
      i_ResultRequest : Bool;
      i_Reset : Bool;
      i_CheckTimeOut : DInt := 10000;
      i_ResultTimeOut : DInt := 10000;
      i_Status : Int;
   END_VAR
   VAR_OUTPUT
      o_CheckTimeOut : Bool;
      o_ResultTimeOut : Bool;
   END_VAR
   VAR_IN_OUT
      ioPLC_MESCheckReq : Bool;
      ioPLC_MESResultReq : Bool;
      ioMES_PLCChecOK : Bool;
      ioMES_PLCChecNG : Bool;
      ioMES_PLCChecDone : Bool;
      ioMES_PLCResultOK : Bool;
      ioMES_PLCResultNG : Bool;
      ioMES_PLCResultDone : Bool;
      ioProductStatus : Int;
   END_VAR
   VAR
      CheckStep : Int;
      ResultStep : Int;
      CheckTimeOut : TON_TIME;
      ResultTimeOut { S7_SetPoint := 'True'} : TON_TIME;
      Pls : Array[0..20] of Bool;
   END_VAR
   VAR_TEMP   // added for the SCL form of the ladder/FBD networks
      _w1 : Bool;
      _w2 : Bool;
      _w3 : Bool;
      _w4 : Bool;
      _w5 : Bool;
      _w6 : Bool;
      _w7 : Bool;
   END_VAR
BEGIN

REGION Network 1: MES Check In Start
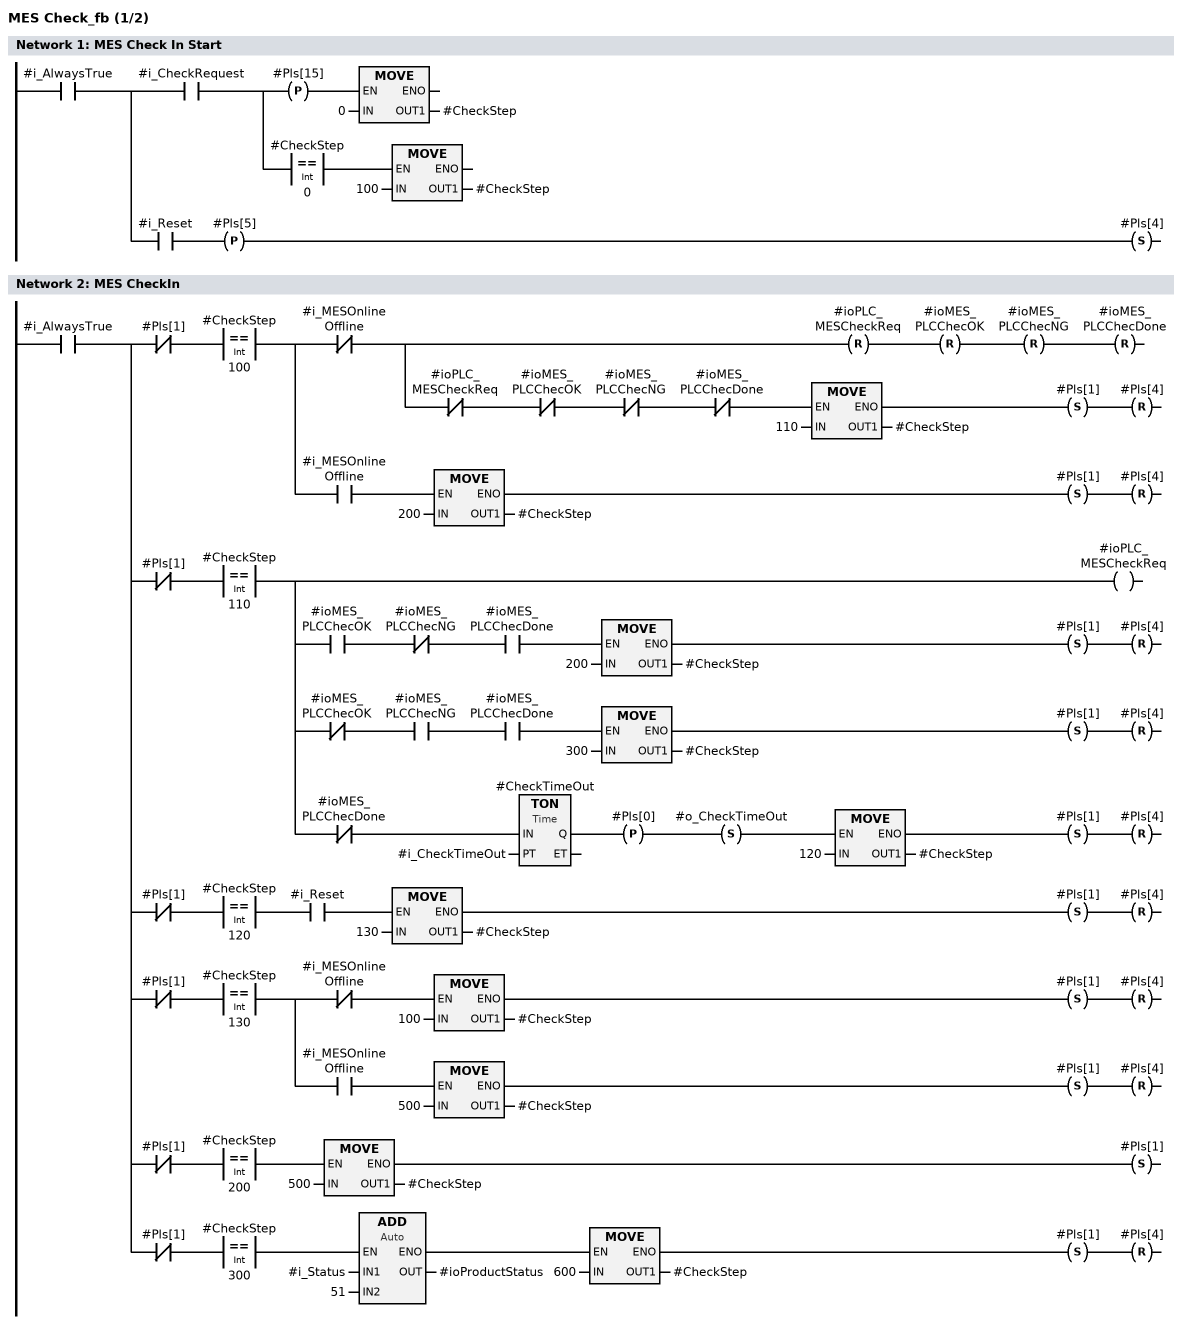
   RUNG wire#powerrail
      Contact( #i_AlwaysTrue )
      wire#w1
      Contact( #i_CheckRequest )
      wire#w2
      P_Trig( #Pls[15] )
      Move(in := 0, out1 => #CheckStep)
   END_RUNG
   RUNG wire#w2
      { S7_Templates := "SrcType := Int" } EQ_Contact(in1 := #CheckStep, in2 := 0)
      Move(in := 100, out1 => #CheckStep)
   END_RUNG
   RUNG wire#w1
      Contact( #i_Reset )
      P_Trig( #Pls[5] )
      S_Coil( #Pls[4] )
   END_RUNG
   // the same network as SCL:
   #_w1 := #i_AlwaysTrue AND #i_CheckRequest;
   #_w2 := #_w1 AND NOT #Pls[15];   // rising edge
   #Pls[15] := #_w1;
   IF #_w2 THEN #CheckStep := 0; END_IF;
   IF #_w1 AND (#CheckStep = 0) THEN #CheckStep := 100; END_IF;
   #_w3 := #i_AlwaysTrue AND #i_Reset;
   #_w4 := #_w3 AND NOT #Pls[5];   // rising edge
   #Pls[5] := #_w3;
   IF #_w4 THEN #Pls[4] := TRUE; END_IF;
END_REGION

REGION Network 2: MES CheckIn
   RUNG wire#powerrail
      Contact( #i_AlwaysTrue )
      wire#w1
      I_Contact( #Pls[1] )
      { S7_Templates := "SrcType := Int" } EQ_Contact(in1 := #CheckStep, in2 := 100)
      wire#w2
      I_Contact( #i_MESOnlineOffline )
      wire#w3
      R_Coil( #ioPLC_MESCheckReq )
      R_Coil( #ioMES_PLCChecOK )
      R_Coil( #ioMES_PLCChecNG )
      R_Coil( #ioMES_PLCChecDone )
   END_RUNG
   RUNG wire#w3
      I_Contact( #ioPLC_MESCheckReq )
      I_Contact( #ioMES_PLCChecOK )
      I_Contact( #ioMES_PLCChecNG )
      I_Contact( #ioMES_PLCChecDone )
      Move(in := 110, out1 => #CheckStep)
      S_Coil( #Pls[1] )
      R_Coil( #Pls[4] )
   END_RUNG
   RUNG wire#w2
      Contact( #i_MESOnlineOffline )
      Move(in := 200, out1 => #CheckStep)
      S_Coil( #Pls[1] )
      R_Coil( #Pls[4] )
   END_RUNG
   RUNG wire#w1
      I_Contact( #Pls[1] )
      { S7_Templates := "SrcType := Int" } EQ_Contact(in1 := #CheckStep, in2 := 110)
      wire#w4
      Coil( #ioPLC_MESCheckReq )
   END_RUNG
   RUNG wire#w4
      Contact( #ioMES_PLCChecOK )
      I_Contact( #ioMES_PLCChecNG )
      Contact( #ioMES_PLCChecDone )
      Move(in := 200, out1 => #CheckStep)
      S_Coil( #Pls[1] )
      R_Coil( #Pls[4] )
   END_RUNG
   RUNG wire#w4
      I_Contact( #ioMES_PLCChecOK )
      Contact( #ioMES_PLCChecNG )
      Contact( #ioMES_PLCChecDone )
      Move(in := 300, out1 => #CheckStep)
      S_Coil( #Pls[1] )
      R_Coil( #Pls[4] )
   END_RUNG
   RUNG wire#w4
      I_Contact( #ioMES_PLCChecDone )
      { S7_Templates := "time_type := Time" } #CheckTimeOut.TON(pt := #i_CheckTimeOut, et =>)
      P_Trig( #Pls[0] )
      S_Coil( #o_CheckTimeOut )
      Move(in := 120, out1 => #CheckStep)
      S_Coil( #Pls[1] )
      R_Coil( #Pls[4] )
   END_RUNG
   RUNG wire#w1
      I_Contact( #Pls[1] )
      { S7_Templates := "SrcType := Int" } EQ_Contact(in1 := #CheckStep, in2 := 120)
      Contact( #i_Reset )
      Move(in := 130, out1 => #CheckStep)
      S_Coil( #Pls[1] )
      R_Coil( #Pls[4] )
   END_RUNG
   RUNG wire#w1
      I_Contact( #Pls[1] )
      { S7_Templates := "SrcType := Int" } EQ_Contact(in1 := #CheckStep, in2 := 130)
      wire#w5
      I_Contact( #i_MESOnlineOffline )
      Move(in := 100, out1 => #CheckStep)
      S_Coil( #Pls[1] )
      R_Coil( #Pls[4] )
   END_RUNG
   RUNG wire#w5
      Contact( #i_MESOnlineOffline )
      Move(in := 500, out1 => #CheckStep)
      S_Coil( #Pls[1] )
      R_Coil( #Pls[4] )
   END_RUNG
   RUNG wire#w1
      I_Contact( #Pls[1] )
      { S7_Templates := "SrcType := Int" } EQ_Contact(in1 := #CheckStep, in2 := 200)
      Move(in := 500, out1 => #CheckStep)
      S_Coil( #Pls[1] )
   END_RUNG
   RUNG wire#w1
      I_Contact( #Pls[1] )
      { S7_Templates := "SrcType := Int" } EQ_Contact(in1 := #CheckStep, in2 := 300)
      Add(in1 := #i_Status, in2 := 51, out => #ioProductStatus)
      Move(in := 600, out1 => #CheckStep)
      S_Coil( #Pls[1] )
      R_Coil( #Pls[4] )
   END_RUNG
   // the same network as SCL:
   #_w1 := #i_AlwaysTrue AND NOT #Pls[1] AND (#CheckStep = 100);
   #_w2 := #_w1 AND NOT #i_MESOnlineOffline;
   IF #_w2 THEN
       #ioPLC_MESCheckReq := FALSE;
       #ioMES_PLCChecOK := FALSE;
       #ioMES_PLCChecNG := FALSE;
       #ioMES_PLCChecDone := FALSE;
   END_IF;
   IF #_w2 AND NOT #ioPLC_MESCheckReq AND NOT #ioMES_PLCChecOK AND NOT #ioMES_PLCChecNG AND NOT #ioMES_PLCChecDone THEN
       #CheckStep := 110;
       #Pls[1] := TRUE;
       #Pls[4] := FALSE;
   END_IF;
   IF #_w1 AND #i_MESOnlineOffline THEN
       #CheckStep := 200;
       #Pls[1] := TRUE;
       #Pls[4] := FALSE;
   END_IF;
   #ioPLC_MESCheckReq := #i_AlwaysTrue AND NOT #Pls[1] AND (#CheckStep = 110);
   IF #ioPLC_MESCheckReq AND #ioMES_PLCChecOK AND NOT #ioMES_PLCChecNG AND #ioMES_PLCChecDone THEN
       #CheckStep := 200;
       #Pls[1] := TRUE;
       #Pls[4] := FALSE;
   END_IF;
   IF #ioPLC_MESCheckReq AND NOT #ioMES_PLCChecOK AND #ioMES_PLCChecNG AND #ioMES_PLCChecDone THEN
       #CheckStep := 300;
       #Pls[1] := TRUE;
       #Pls[4] := FALSE;
   END_IF;
   #CheckTimeOut(IN := #ioPLC_MESCheckReq AND NOT #ioMES_PLCChecDone, PT := #i_CheckTimeOut);   // TON
   #_w3 := #CheckTimeOut.Q AND NOT #Pls[0];   // rising edge
   #Pls[0] := #CheckTimeOut.Q;
   IF #_w3 THEN
       #o_CheckTimeOut := TRUE;
       #CheckStep := 120;
       #Pls[1] := TRUE;
       #Pls[4] := FALSE;
   END_IF;
   #_w4 := #i_AlwaysTrue AND NOT #Pls[1] AND (#CheckStep = 120) AND #i_Reset;
   IF #_w4 THEN
       #CheckStep := 130;
       #Pls[1] := TRUE;
       #Pls[4] := FALSE;
   END_IF;
   #_w5 := #i_AlwaysTrue AND NOT #Pls[1] AND (#CheckStep = 130);
   IF #_w5 AND NOT #i_MESOnlineOffline THEN
       #CheckStep := 100;
       #Pls[1] := TRUE;
       #Pls[4] := FALSE;
   END_IF;
   IF #_w5 AND #i_MESOnlineOffline THEN
       #CheckStep := 500;
       #Pls[1] := TRUE;
       #Pls[4] := FALSE;
   END_IF;
   #_w6 := #i_AlwaysTrue AND NOT #Pls[1] AND (#CheckStep = 200);
   IF #_w6 THEN
       #CheckStep := 500;
       #Pls[1] := TRUE;
   END_IF;
   IF #i_AlwaysTrue AND NOT #Pls[1] AND (#CheckStep = 300) THEN #ioProductStatus := #i_Status + 51; END_IF;
   #_w7 := #i_AlwaysTrue AND NOT #Pls[1] AND (#CheckStep = 300);
   IF #_w7 THEN
       #CheckStep := 600;
       #Pls[1] := TRUE;
       #Pls[4] := FALSE;
   END_IF;
END_REGION

REGION Network 4: MES Check Out Start
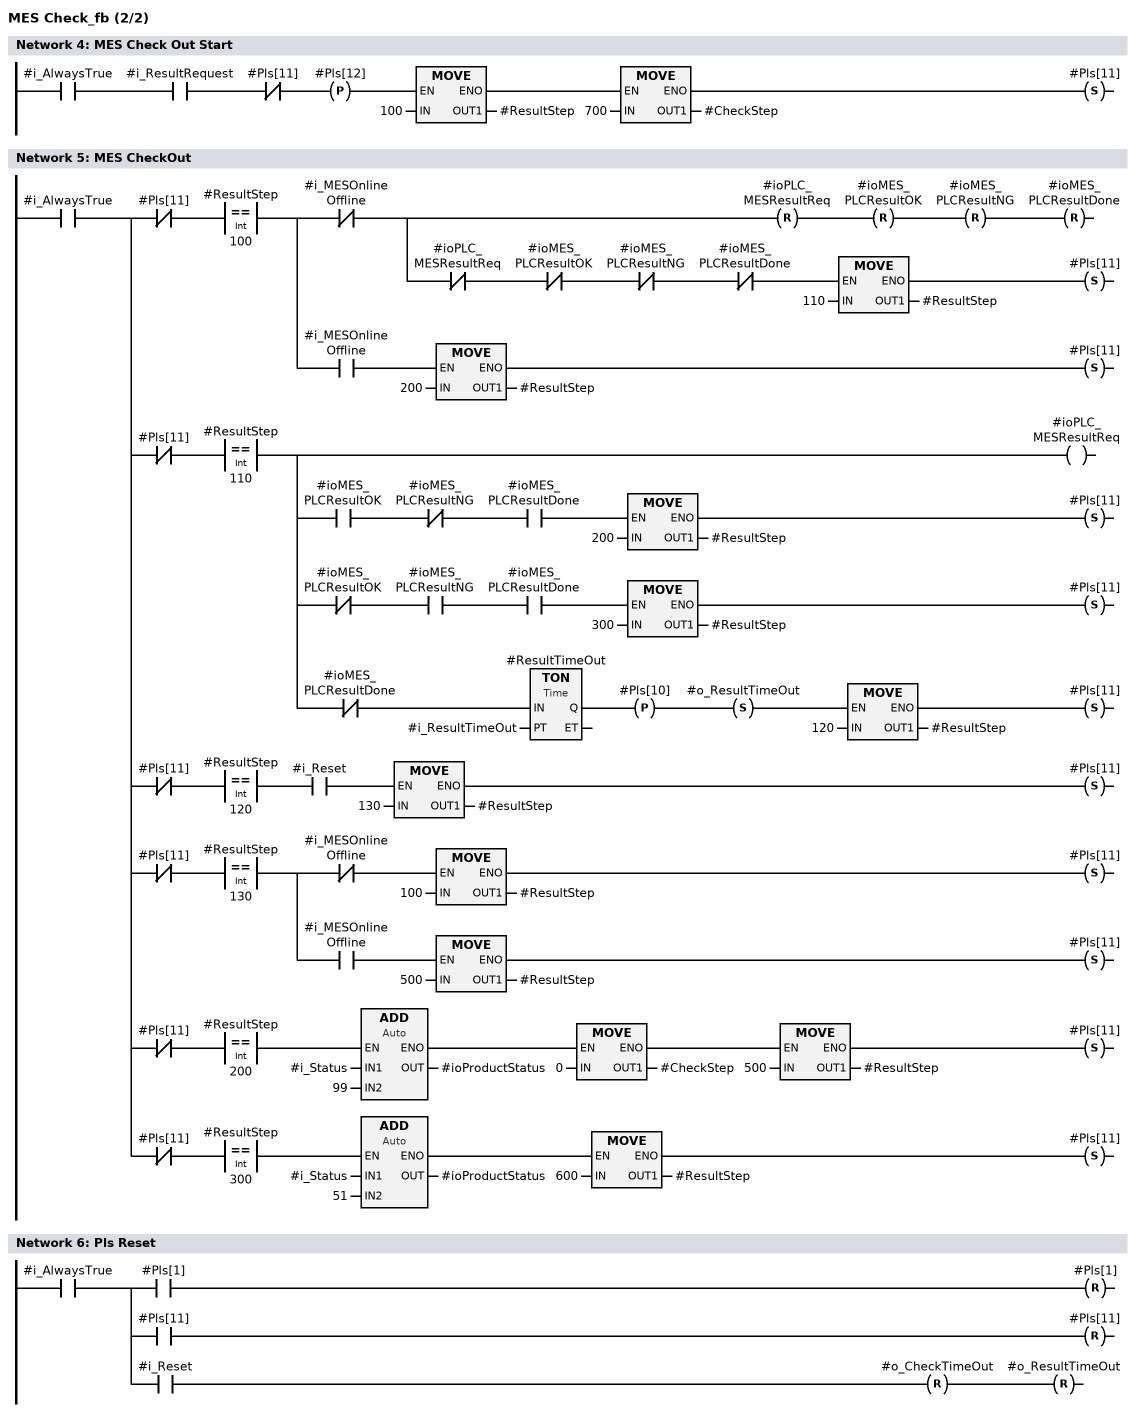
   RUNG wire#powerrail
      Contact( #i_AlwaysTrue )
      Contact( #i_ResultRequest )
      I_Contact( #Pls[11] )
      P_Trig( #Pls[12] )
      Move(in := 100, out1 => #ResultStep)
      Move(in := 700, out1 => #CheckStep)
      S_Coil( #Pls[11] )
   END_RUNG
   // the same network as SCL:
   #_w1 := #i_AlwaysTrue AND #i_ResultRequest AND NOT #Pls[11];
   #_w2 := #_w1 AND NOT #Pls[12];   // rising edge
   #Pls[12] := #_w1;
   IF #_w2 THEN
       #ResultStep := 100;
       #CheckStep := 700;
       #Pls[11] := TRUE;
   END_IF;
END_REGION

REGION Network 5: MES CheckOut
   RUNG wire#powerrail
      Contact( #i_AlwaysTrue )
      wire#w1
      I_Contact( #Pls[11] )
      { S7_Templates := "SrcType := Int" } EQ_Contact(in1 := #ResultStep, in2 := 100)
      wire#w2
      I_Contact( #i_MESOnlineOffline )
      wire#w3
      R_Coil( #ioPLC_MESResultReq )
      R_Coil( #ioMES_PLCResultOK )
      R_Coil( #ioMES_PLCResultNG )
      R_Coil( #ioMES_PLCResultDone )
   END_RUNG
   RUNG wire#w3
      I_Contact( #ioPLC_MESResultReq )
      I_Contact( #ioMES_PLCResultOK )
      I_Contact( #ioMES_PLCResultNG )
      I_Contact( #ioMES_PLCResultDone )
      Move(in := 110, out1 => #ResultStep)
      S_Coil( #Pls[11] )
   END_RUNG
   RUNG wire#w2
      Contact( #i_MESOnlineOffline )
      Move(in := 200, out1 => #ResultStep)
      S_Coil( #Pls[11] )
   END_RUNG
   RUNG wire#w1
      I_Contact( #Pls[11] )
      { S7_Templates := "SrcType := Int" } EQ_Contact(in1 := #ResultStep, in2 := 110)
      wire#w4
      Coil( #ioPLC_MESResultReq )
   END_RUNG
   RUNG wire#w4
      Contact( #ioMES_PLCResultOK )
      I_Contact( #ioMES_PLCResultNG )
      Contact( #ioMES_PLCResultDone )
      Move(in := 200, out1 => #ResultStep)
      S_Coil( #Pls[11] )
   END_RUNG
   RUNG wire#w4
      I_Contact( #ioMES_PLCResultOK )
      Contact( #ioMES_PLCResultNG )
      Contact( #ioMES_PLCResultDone )
      Move(in := 300, out1 => #ResultStep)
      S_Coil( #Pls[11] )
   END_RUNG
   RUNG wire#w4
      I_Contact( #ioMES_PLCResultDone )
      { S7_Templates := "time_type := Time" } #ResultTimeOut.TON(pt := #i_ResultTimeOut, et =>)
      P_Trig( #Pls[10] )
      S_Coil( #o_ResultTimeOut )
      Move(in := 120, out1 => #ResultStep)
      S_Coil( #Pls[11] )
   END_RUNG
   RUNG wire#w1
      I_Contact( #Pls[11] )
      { S7_Templates := "SrcType := Int" } EQ_Contact(in1 := #ResultStep, in2 := 120)
      Contact( #i_Reset )
      Move(in := 130, out1 => #ResultStep)
      S_Coil( #Pls[11] )
   END_RUNG
   RUNG wire#w1
      I_Contact( #Pls[11] )
      { S7_Templates := "SrcType := Int" } EQ_Contact(in1 := #ResultStep, in2 := 130)
      wire#w5
      I_Contact( #i_MESOnlineOffline )
      Move(in := 100, out1 => #ResultStep)
      S_Coil( #Pls[11] )
   END_RUNG
   RUNG wire#w5
      Contact( #i_MESOnlineOffline )
      Move(in := 500, out1 => #ResultStep)
      S_Coil( #Pls[11] )
   END_RUNG
   RUNG wire#w1
      I_Contact( #Pls[11] )
      { S7_Templates := "SrcType := Int" } EQ_Contact(in1 := #ResultStep, in2 := 200)
      Add(in1 := #i_Status, in2 := 99, out => #ioProductStatus)
      Move(in := 0, out1 => #CheckStep)
      Move(in := 500, out1 => #ResultStep)
      S_Coil( #Pls[11] )
   END_RUNG
   RUNG wire#w1
      I_Contact( #Pls[11] )
      { S7_Templates := "SrcType := Int" } EQ_Contact(in1 := #ResultStep, in2 := 300)
      Add(in1 := #i_Status, in2 := 51, out => #ioProductStatus)
      Move(in := 600, out1 => #ResultStep)
      S_Coil( #Pls[11] )
   END_RUNG
   // the same network as SCL:
   #_w1 := #i_AlwaysTrue AND NOT #Pls[11] AND (#ResultStep = 100);
   #_w2 := #_w1 AND NOT #i_MESOnlineOffline;
   IF #_w2 THEN
       #ioPLC_MESResultReq := FALSE;
       #ioMES_PLCResultOK := FALSE;
       #ioMES_PLCResultNG := FALSE;
       #ioMES_PLCResultDone := FALSE;
   END_IF;
   IF #_w2 AND NOT #ioPLC_MESResultReq AND NOT #ioMES_PLCResultOK AND NOT #ioMES_PLCResultNG AND NOT #ioMES_PLCResultDone THEN
       #ResultStep := 110;
       #Pls[11] := TRUE;
   END_IF;
   IF #_w1 AND #i_MESOnlineOffline THEN
       #ResultStep := 200;
       #Pls[11] := TRUE;
   END_IF;
   #ioPLC_MESResultReq := #i_AlwaysTrue AND NOT #Pls[11] AND (#ResultStep = 110);
   IF #ioPLC_MESResultReq AND #ioMES_PLCResultOK AND NOT #ioMES_PLCResultNG AND #ioMES_PLCResultDone THEN
       #ResultStep := 200;
       #Pls[11] := TRUE;
   END_IF;
   IF #ioPLC_MESResultReq AND NOT #ioMES_PLCResultOK AND #ioMES_PLCResultNG AND #ioMES_PLCResultDone THEN
       #ResultStep := 300;
       #Pls[11] := TRUE;
   END_IF;
   #ResultTimeOut(IN := #ioPLC_MESResultReq AND NOT #ioMES_PLCResultDone, PT := #i_ResultTimeOut);   // TON
   #_w3 := #ResultTimeOut.Q AND NOT #Pls[10];   // rising edge
   #Pls[10] := #ResultTimeOut.Q;
   IF #_w3 THEN
       #o_ResultTimeOut := TRUE;
       #ResultStep := 120;
       #Pls[11] := TRUE;
   END_IF;
   #_w4 := #i_AlwaysTrue AND NOT #Pls[11] AND (#ResultStep = 120) AND #i_Reset;
   IF #_w4 THEN
       #ResultStep := 130;
       #Pls[11] := TRUE;
   END_IF;
   #_w5 := #i_AlwaysTrue AND NOT #Pls[11] AND (#ResultStep = 130);
   IF #_w5 AND NOT #i_MESOnlineOffline THEN
       #ResultStep := 100;
       #Pls[11] := TRUE;
   END_IF;
   IF #_w5 AND #i_MESOnlineOffline THEN
       #ResultStep := 500;
       #Pls[11] := TRUE;
   END_IF;
   IF #i_AlwaysTrue AND NOT #Pls[11] AND (#ResultStep = 200) THEN
       #ioProductStatus := #i_Status + 99;
       #CheckStep := 0;
   END_IF;
   #_w6 := #i_AlwaysTrue AND NOT #Pls[11] AND (#ResultStep = 200);
   IF #_w6 THEN
       #ResultStep := 500;
       #Pls[11] := TRUE;
   END_IF;
   IF #i_AlwaysTrue AND NOT #Pls[11] AND (#ResultStep = 300) THEN #ioProductStatus := #i_Status + 51; END_IF;
   #_w7 := #i_AlwaysTrue AND NOT #Pls[11] AND (#ResultStep = 300);
   IF #_w7 THEN
       #ResultStep := 600;
       #Pls[11] := TRUE;
   END_IF;
END_REGION

REGION Network 6: Pls Reset
   RUNG wire#powerrail
      Contact( #i_AlwaysTrue )
      wire#w1
      Contact( #Pls[1] )
      R_Coil( #Pls[1] )
   END_RUNG
   RUNG wire#w1
      Contact( #Pls[11] )
      R_Coil( #Pls[11] )
   END_RUNG
   RUNG wire#w1
      Contact( #i_Reset )
      R_Coil( #o_CheckTimeOut )
      R_Coil( #o_ResultTimeOut )
   END_RUNG
   // the same network as SCL:
   IF #i_AlwaysTrue AND #Pls[1] THEN #Pls[1] := FALSE; END_IF;
   IF #i_AlwaysTrue AND #Pls[11] THEN #Pls[11] := FALSE; END_IF;
   IF #i_AlwaysTrue AND #i_Reset THEN
       #o_CheckTimeOut := FALSE;
       #o_ResultTimeOut := FALSE;
   END_IF;
END_REGION
END_FUNCTION_BLOCK

FUNCTION_BLOCK "ST10_CountCycleTimeMain"   // FB1009, LAD
{ S7_Optimized_Access := 'TRUE' }
VERSION : 0.1
// stored: AutoNumber false, IsIECCheckEnabled false, IsRetainMemResEnabled false, MemoryReserve 100, SetENOAutomatically false, UDAEnableTagReadback false
   VAR_INPUT
      iAlwaysOn : Bool;
      iRun : Bool;
      iManualMode : Bool;
      iAutoMode : Bool;
      iAutoRunning : Bool;
   END_VAR
   VAR
      MianCountCycleTime { S7_SetPoint := 'True'} : "Count_CycleTime";
      PM1CountCycleTime { S7_SetPoint := 'True'} : "Count_CycleTime_V3";
      PM2CountCycleTime { S7_SetPoint := 'True'} : "Count_CycleTime_V3";
      PM3CountCycleTime { S7_SetPoint := 'True'} : "Count_CycleTime_V3";
      PM4CountCycleTime { S7_SetPoint := 'True'} : "Count_CycleTime_V3";
      PM5CountCycleTime { S7_SetPoint := 'True'} : "Count_CycleTime_V3";
      PM6CountCycleTime { S7_SetPoint := 'True'} : "Count_CycleTime_V3";
      PM7CountCycleTime { S7_SetPoint := 'True'} : "Count_CycleTime_V3";
      PM8CountCycleTime { S7_SetPoint := 'True'} : "Count_CycleTime_V3";
      PM9CountCycleTime { S7_SetPoint := 'True'} : "Count_CycleTime_V3";
      PM10CountCycleTime { S7_SetPoint := 'True'} : "Count_CycleTime_V3";
      PM11CountCycleTime { S7_SetPoint := 'True'} : "Count_CycleTime_V3";
      PM12CountCycleTime { S7_SetPoint := 'True'} : "Count_CycleTime_V3";
      PM13CountCycleTime { S7_SetPoint := 'True'} : "Count_CycleTime_V3";
      PM14CountCycleTime { S7_SetPoint := 'True'} : "Count_CycleTime_V3";
      PM15CountCycleTime { S7_SetPoint := 'True'} : "Count_CycleTime_V3";
      PM16CountCycleTime { S7_SetPoint := 'True'} : "Count_CycleTime_V3";
      PM17CountCycleTime { S7_SetPoint := 'True'} : "Count_CycleTime_V3";
      PM18CountCycleTime { S7_SetPoint := 'True'} : "Count_CycleTime_V3";
      PM19CountCycleTime { S7_SetPoint := 'True'} : "Count_CycleTime_V3";
      PM20CountCycleTime { S7_SetPoint := 'True'} : "Count_CycleTime_V3";
      PM21CountCycleTime { S7_SetPoint := 'True'} : "Count_CycleTime_V3";
      PM22CountCycleTime { S7_SetPoint := 'True'} : "Count_CycleTime_V3";
      PM23CountCycleTime { S7_SetPoint := 'True'} : "Count_CycleTime_V3";
      PM24CountCycleTime { S7_SetPoint := 'True'} : "Count_CycleTime_V3";
      PM25CountCycleTime { S7_SetPoint := 'True'} : "Count_CycleTime_V3";
      PM26CountCycleTime { S7_SetPoint := 'True'} : "Count_CycleTime_V3";
      PM27CountCycleTime { S7_SetPoint := 'True'} : "Count_CycleTime_V3";
      PM28CountCycleTime { S7_SetPoint := 'True'} : "Count_CycleTime_V3";
      PM29CountCycleTime { S7_SetPoint := 'True'} : "Count_CycleTime_V3";
      PM30CountCycleTime { S7_SetPoint := 'True'} : "Count_CycleTime_V3";
   END_VAR
BEGIN

REGION Network 1: Mian Count & CycleTime
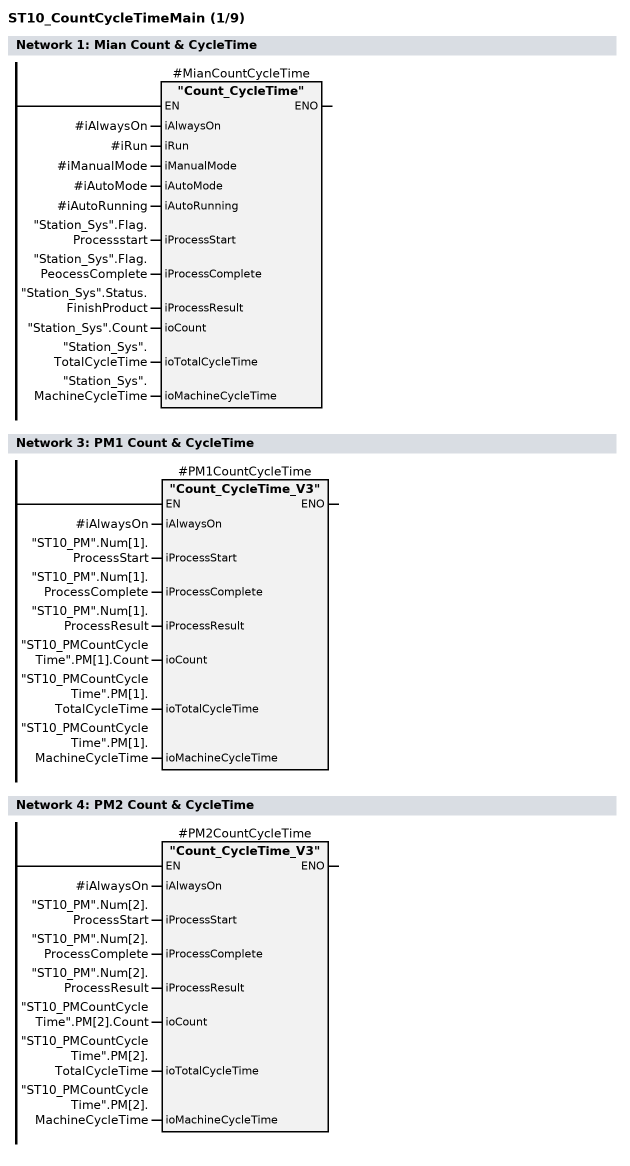
   RUNG wire#powerrail
      #MianCountCycleTime(iAlwaysOn := #iAlwaysOn, iRun := #iRun, iManualMode := #iManualMode, iAutoMode := #iAutoMode, iAutoRunning := #iAutoRunning, iProcessStart := "Station_Sys".Flag.Processstart, iProcessComplete := "Station_Sys".Flag.PeocessComplete, iProcessResult := "Station_Sys".Status.FinishProduct, ioCount := "Station_Sys".Count, ioTotalCycleTime := "Station_Sys".TotalCycleTime, ioMachineCycleTime := "Station_Sys".MachineCycleTime)
   END_RUNG
   // the same network as SCL:
   #MianCountCycleTime(iAlwaysOn := #iAlwaysOn,   // "Count_CycleTime"
                       iRun := #iRun,
                       iManualMode := #iManualMode,
                       iAutoMode := #iAutoMode,
                       iAutoRunning := #iAutoRunning,
                       iProcessStart := "Station_Sys".Flag.Processstart,
                       iProcessComplete := "Station_Sys".Flag.PeocessComplete,
                       iProcessResult := "Station_Sys".Status.FinishProduct,
                       ioCount := "Station_Sys".Count,
                       ioTotalCycleTime := "Station_Sys".TotalCycleTime,
                       ioMachineCycleTime := "Station_Sys".MachineCycleTime);
END_REGION

REGION Network 2 (SCL)
   "ST10_PMCountCycleTime".PM[1].Num := 1;
   "ST10_PMCountCycleTime".PM[2].Num := 2;
   "ST10_PMCountCycleTime".PM[3].Num := 3;
   "ST10_PMCountCycleTime".PM[4].Num := 4;
   "ST10_PMCountCycleTime".PM[5].Num := 5;
   "ST10_PMCountCycleTime".PM[6].Num := 6;
   "ST10_PMCountCycleTime".PM[7].Num := 7;
   "ST10_PMCountCycleTime".PM[8].Num := 8;
   "ST10_PMCountCycleTime".PM[9].Num := 9;
   "ST10_PMCountCycleTime".PM[10].Num := 10;
   "ST10_PMCountCycleTime".PM[11].Num := 11;
   "ST10_PMCountCycleTime".PM[12].Num := 12;
   "ST10_PMCountCycleTime".PM[13].Num := 13;
   "ST10_PMCountCycleTime".PM[14].Num := 14;
   "ST10_PMCountCycleTime".PM[15].Num := 15;
   "ST10_PMCountCycleTime".PM[16].Num := 16;
   "ST10_PMCountCycleTime".PM[17].Num := 17;
   "ST10_PMCountCycleTime".PM[18].Num := 18;
   "ST10_PMCountCycleTime".PM[19].Num := 19;
   "ST10_PMCountCycleTime".PM[20].Num := 20;
   "ST10_PMCountCycleTime".PM[21].Num := 21;
   "ST10_PMCountCycleTime".PM[22].Num := 22;
   "ST10_PMCountCycleTime".PM[23].Num := 23;
   "ST10_PMCountCycleTime".PM[24].Num := 24;
   "ST10_PMCountCycleTime".PM[25].Num := 25;
   // "ST70_PMCountCycleTime".PM[5].Num := 5;
   // "ST70_PMCountCycleTime".PM[6].Num := 6;
   // "ST70_PMCountCycleTime".PM[7].Num := 7;
   // "ST70_PMCountCycleTime".PM[8].Num := 8;
   // "ST70_PMCountCycleTime".PM[9].Num := 9;
   // "ST70_PMCountCycleTime".PM[10].Num := 10;
   //TEST
   (*
   "ST10_PMCountCycleTime".PM[1].Count.OK[0] := 10;
   "ST10_PMCountCycleTime".PM[2].Count.OK[0] := 20;
   "ST10_PMCountCycleTime".PM[3].Count.OK[0] := 30;
   "ST10_PMCountCycleTime".PM[4].Count.OK[0] := 40;
   "ST10_PMCountCycleTime".PM[5].Count.OK[0] := 50;
   "ST10_PMCountCycleTime".PM[6].Count.OK[0] := 60;
   "ST10_PMCountCycleTime".PM[7].Count.OK[0] := 70;
   "ST10_PMCountCycleTime".PM[8].Count.OK[0] := 80;
   "ST10_PMCountCycleTime".PM[9].Count.OK[0] := 90;
   "ST10_PMCountCycleTime".PM[10].Count.OK[0] := 100;

   "ST10_PMCountCycleTime".PM[1].TotalCycleTime.No[0] := 100;
   "ST10_PMCountCycleTime".PM[2].TotalCycleTime.No[0] := 200;
   "ST10_PMCountCycleTime".PM[3].TotalCycleTime.No[0] := 300;
   "ST10_PMCountCycleTime".PM[4].TotalCycleTime.No[0] := 400;
   "ST10_PMCountCycleTime".PM[5].TotalCycleTime.No[0] := 500;
   "ST10_PMCountCycleTime".PM[6].TotalCycleTime.No[0] := 600;
   "ST10_PMCountCycleTime".PM[7].TotalCycleTime.No[0] := 700;
   "ST10_PMCountCycleTime".PM[8].TotalCycleTime.No[0] := 800;
   "ST10_PMCountCycleTime".PM[9].TotalCycleTime.No[0] := 900;
   "ST10_PMCountCycleTime".PM[10].TotalCycleTime.No[0] := 1000;

   "ST10_PMCountCycleTime".PM[1].MachineCycleTime.No[0] := 110;
   "ST10_PMCountCycleTime".PM[2].MachineCycleTime.No[0] := 220;
   "ST10_PMCountCycleTime".PM[3].MachineCycleTime.No[0] := 330;
   "ST10_PMCountCycleTime".PM[4].MachineCycleTime.No[0] := 440;
   "ST10_PMCountCycleTime".PM[5].MachineCycleTime.No[0] := 550;
   "ST10_PMCountCycleTime".PM[6].MachineCycleTime.No[0] := 660;
   "ST10_PMCountCycleTime".PM[7].MachineCycleTime.No[0] := 770;
   "ST10_PMCountCycleTime".PM[8].MachineCycleTime.No[0] := 880;
   "ST10_PMCountCycleTime".PM[9].MachineCycleTime.No[0] := 990;
   "ST10_PMCountCycleTime".PM[10].MachineCycleTime.No[0] := 1010;
   *)
END_REGION

REGION Network 3: PM1 Count & CycleTime
   RUNG wire#powerrail
      #PM1CountCycleTime(iAlwaysOn := #iAlwaysOn, iProcessStart := "ST10_PM".Num[1].ProcessStart, iProcessComplete := "ST10_PM".Num[1].ProcessComplete, iProcessResult := "ST10_PM".Num[1].ProcessResult, ioCount := "ST10_PMCountCycleTime".PM[1].Count, ioTotalCycleTime := "ST10_PMCountCycleTime".PM[1].TotalCycleTime, ioMachineCycleTime := "ST10_PMCountCycleTime".PM[1].MachineCycleTime)
   END_RUNG
   // the same network as SCL:
   #PM1CountCycleTime(iAlwaysOn := #iAlwaysOn,   // "Count_CycleTime_V3"
                      iProcessStart := "ST10_PM".Num[1].ProcessStart,
                      iProcessComplete := "ST10_PM".Num[1].ProcessComplete,
                      iProcessResult := "ST10_PM".Num[1].ProcessResult,
                      ioCount := "ST10_PMCountCycleTime".PM[1].Count,
                      ioTotalCycleTime := "ST10_PMCountCycleTime".PM[1].TotalCycleTime,
                      ioMachineCycleTime := "ST10_PMCountCycleTime".PM[1].MachineCycleTime);
END_REGION

REGION Network 4: PM2 Count & CycleTime
   RUNG wire#powerrail
      #PM2CountCycleTime(iAlwaysOn := #iAlwaysOn, iProcessStart := "ST10_PM".Num[2].ProcessStart, iProcessComplete := "ST10_PM".Num[2].ProcessComplete, iProcessResult := "ST10_PM".Num[2].ProcessResult, ioCount := "ST10_PMCountCycleTime".PM[2].Count, ioTotalCycleTime := "ST10_PMCountCycleTime".PM[2].TotalCycleTime, ioMachineCycleTime := "ST10_PMCountCycleTime".PM[2].MachineCycleTime)
   END_RUNG
   // the same network as SCL:
   #PM2CountCycleTime(iAlwaysOn := #iAlwaysOn,   // "Count_CycleTime_V3"
                      iProcessStart := "ST10_PM".Num[2].ProcessStart,
                      iProcessComplete := "ST10_PM".Num[2].ProcessComplete,
                      iProcessResult := "ST10_PM".Num[2].ProcessResult,
                      ioCount := "ST10_PMCountCycleTime".PM[2].Count,
                      ioTotalCycleTime := "ST10_PMCountCycleTime".PM[2].TotalCycleTime,
                      ioMachineCycleTime := "ST10_PMCountCycleTime".PM[2].MachineCycleTime);
END_REGION

REGION Network 5: PM3 Count & CycleTime
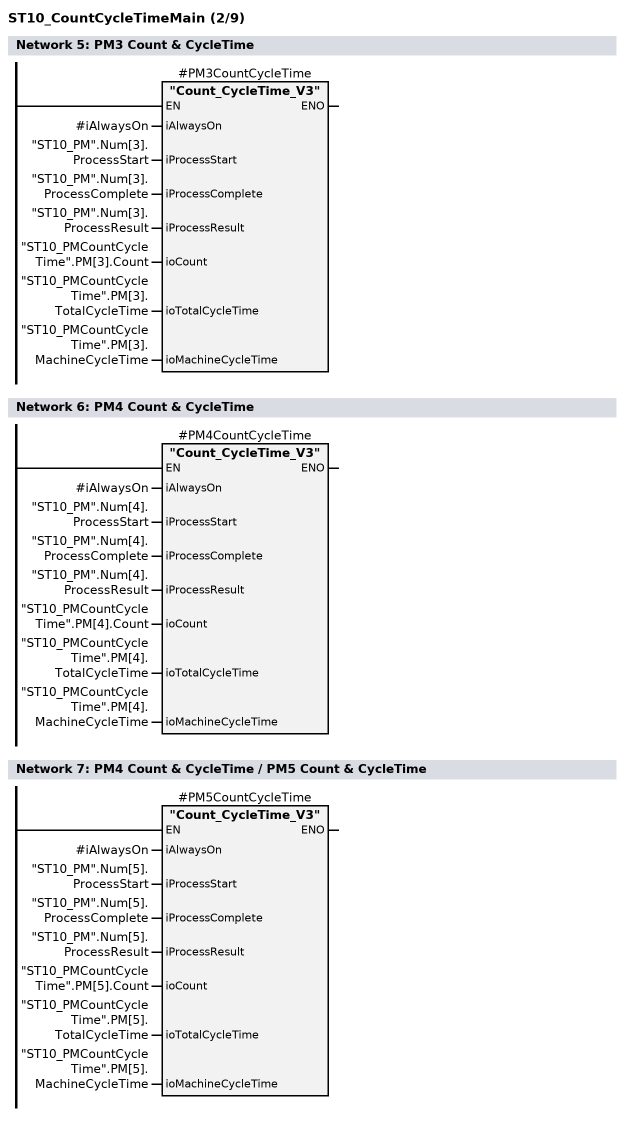
   RUNG wire#powerrail
      #PM3CountCycleTime(iAlwaysOn := #iAlwaysOn, iProcessStart := "ST10_PM".Num[3].ProcessStart, iProcessComplete := "ST10_PM".Num[3].ProcessComplete, iProcessResult := "ST10_PM".Num[3].ProcessResult, ioCount := "ST10_PMCountCycleTime".PM[3].Count, ioTotalCycleTime := "ST10_PMCountCycleTime".PM[3].TotalCycleTime, ioMachineCycleTime := "ST10_PMCountCycleTime".PM[3].MachineCycleTime)
   END_RUNG
   // the same network as SCL:
   #PM3CountCycleTime(iAlwaysOn := #iAlwaysOn,   // "Count_CycleTime_V3"
                      iProcessStart := "ST10_PM".Num[3].ProcessStart,
                      iProcessComplete := "ST10_PM".Num[3].ProcessComplete,
                      iProcessResult := "ST10_PM".Num[3].ProcessResult,
                      ioCount := "ST10_PMCountCycleTime".PM[3].Count,
                      ioTotalCycleTime := "ST10_PMCountCycleTime".PM[3].TotalCycleTime,
                      ioMachineCycleTime := "ST10_PMCountCycleTime".PM[3].MachineCycleTime);
END_REGION

REGION Network 6: PM4 Count & CycleTime
   RUNG wire#powerrail
      #PM4CountCycleTime(iAlwaysOn := #iAlwaysOn, iProcessStart := "ST10_PM".Num[4].ProcessStart, iProcessComplete := "ST10_PM".Num[4].ProcessComplete, iProcessResult := "ST10_PM".Num[4].ProcessResult, ioCount := "ST10_PMCountCycleTime".PM[4].Count, ioTotalCycleTime := "ST10_PMCountCycleTime".PM[4].TotalCycleTime, ioMachineCycleTime := "ST10_PMCountCycleTime".PM[4].MachineCycleTime)
   END_RUNG
   // the same network as SCL:
   #PM4CountCycleTime(iAlwaysOn := #iAlwaysOn,   // "Count_CycleTime_V3"
                      iProcessStart := "ST10_PM".Num[4].ProcessStart,
                      iProcessComplete := "ST10_PM".Num[4].ProcessComplete,
                      iProcessResult := "ST10_PM".Num[4].ProcessResult,
                      ioCount := "ST10_PMCountCycleTime".PM[4].Count,
                      ioTotalCycleTime := "ST10_PMCountCycleTime".PM[4].TotalCycleTime,
                      ioMachineCycleTime := "ST10_PMCountCycleTime".PM[4].MachineCycleTime);
END_REGION

REGION Network 7: PM4 Count & CycleTime / PM5 Count & CycleTime
   RUNG wire#powerrail
      #PM5CountCycleTime(iAlwaysOn := #iAlwaysOn, iProcessStart := "ST10_PM".Num[5].ProcessStart, iProcessComplete := "ST10_PM".Num[5].ProcessComplete, iProcessResult := "ST10_PM".Num[5].ProcessResult, ioCount := "ST10_PMCountCycleTime".PM[5].Count, ioTotalCycleTime := "ST10_PMCountCycleTime".PM[5].TotalCycleTime, ioMachineCycleTime := "ST10_PMCountCycleTime".PM[5].MachineCycleTime)
   END_RUNG
   // the same network as SCL:
   #PM5CountCycleTime(iAlwaysOn := #iAlwaysOn,   // "Count_CycleTime_V3"
                      iProcessStart := "ST10_PM".Num[5].ProcessStart,
                      iProcessComplete := "ST10_PM".Num[5].ProcessComplete,
                      iProcessResult := "ST10_PM".Num[5].ProcessResult,
                      ioCount := "ST10_PMCountCycleTime".PM[5].Count,
                      ioTotalCycleTime := "ST10_PMCountCycleTime".PM[5].TotalCycleTime,
                      ioMachineCycleTime := "ST10_PMCountCycleTime".PM[5].MachineCycleTime);
END_REGION

REGION Network 8: PM4 Count & CycleTime / PM6 Count & CycleTime
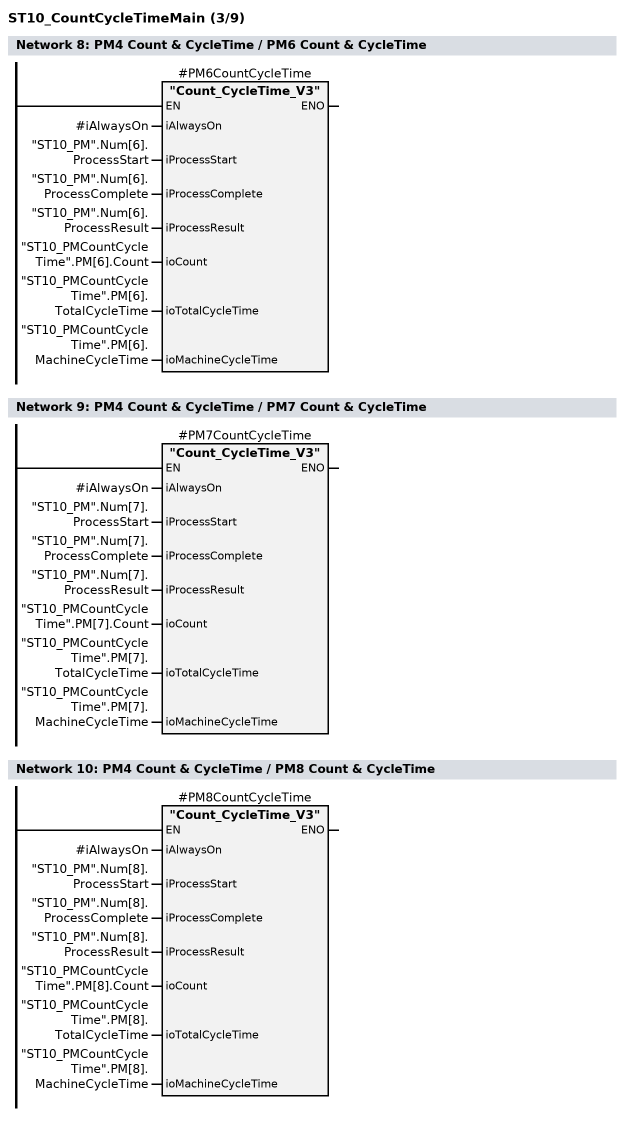
   RUNG wire#powerrail
      #PM6CountCycleTime(iAlwaysOn := #iAlwaysOn, iProcessStart := "ST10_PM".Num[6].ProcessStart, iProcessComplete := "ST10_PM".Num[6].ProcessComplete, iProcessResult := "ST10_PM".Num[6].ProcessResult, ioCount := "ST10_PMCountCycleTime".PM[6].Count, ioTotalCycleTime := "ST10_PMCountCycleTime".PM[6].TotalCycleTime, ioMachineCycleTime := "ST10_PMCountCycleTime".PM[6].MachineCycleTime)
   END_RUNG
   // the same network as SCL:
   #PM6CountCycleTime(iAlwaysOn := #iAlwaysOn,   // "Count_CycleTime_V3"
                      iProcessStart := "ST10_PM".Num[6].ProcessStart,
                      iProcessComplete := "ST10_PM".Num[6].ProcessComplete,
                      iProcessResult := "ST10_PM".Num[6].ProcessResult,
                      ioCount := "ST10_PMCountCycleTime".PM[6].Count,
                      ioTotalCycleTime := "ST10_PMCountCycleTime".PM[6].TotalCycleTime,
                      ioMachineCycleTime := "ST10_PMCountCycleTime".PM[6].MachineCycleTime);
END_REGION

REGION Network 9: PM4 Count & CycleTime / PM7 Count & CycleTime
   RUNG wire#powerrail
      #PM7CountCycleTime(iAlwaysOn := #iAlwaysOn, iProcessStart := "ST10_PM".Num[7].ProcessStart, iProcessComplete := "ST10_PM".Num[7].ProcessComplete, iProcessResult := "ST10_PM".Num[7].ProcessResult, ioCount := "ST10_PMCountCycleTime".PM[7].Count, ioTotalCycleTime := "ST10_PMCountCycleTime".PM[7].TotalCycleTime, ioMachineCycleTime := "ST10_PMCountCycleTime".PM[7].MachineCycleTime)
   END_RUNG
   // the same network as SCL:
   #PM7CountCycleTime(iAlwaysOn := #iAlwaysOn,   // "Count_CycleTime_V3"
                      iProcessStart := "ST10_PM".Num[7].ProcessStart,
                      iProcessComplete := "ST10_PM".Num[7].ProcessComplete,
                      iProcessResult := "ST10_PM".Num[7].ProcessResult,
                      ioCount := "ST10_PMCountCycleTime".PM[7].Count,
                      ioTotalCycleTime := "ST10_PMCountCycleTime".PM[7].TotalCycleTime,
                      ioMachineCycleTime := "ST10_PMCountCycleTime".PM[7].MachineCycleTime);
END_REGION

REGION Network 10: PM4 Count & CycleTime / PM8 Count & CycleTime
   RUNG wire#powerrail
      #PM8CountCycleTime(iAlwaysOn := #iAlwaysOn, iProcessStart := "ST10_PM".Num[8].ProcessStart, iProcessComplete := "ST10_PM".Num[8].ProcessComplete, iProcessResult := "ST10_PM".Num[8].ProcessResult, ioCount := "ST10_PMCountCycleTime".PM[8].Count, ioTotalCycleTime := "ST10_PMCountCycleTime".PM[8].TotalCycleTime, ioMachineCycleTime := "ST10_PMCountCycleTime".PM[8].MachineCycleTime)
   END_RUNG
   // the same network as SCL:
   #PM8CountCycleTime(iAlwaysOn := #iAlwaysOn,   // "Count_CycleTime_V3"
                      iProcessStart := "ST10_PM".Num[8].ProcessStart,
                      iProcessComplete := "ST10_PM".Num[8].ProcessComplete,
                      iProcessResult := "ST10_PM".Num[8].ProcessResult,
                      ioCount := "ST10_PMCountCycleTime".PM[8].Count,
                      ioTotalCycleTime := "ST10_PMCountCycleTime".PM[8].TotalCycleTime,
                      ioMachineCycleTime := "ST10_PMCountCycleTime".PM[8].MachineCycleTime);
END_REGION

REGION Network 11: PM4 Count & CycleTime / PM9 Count & CycleTime
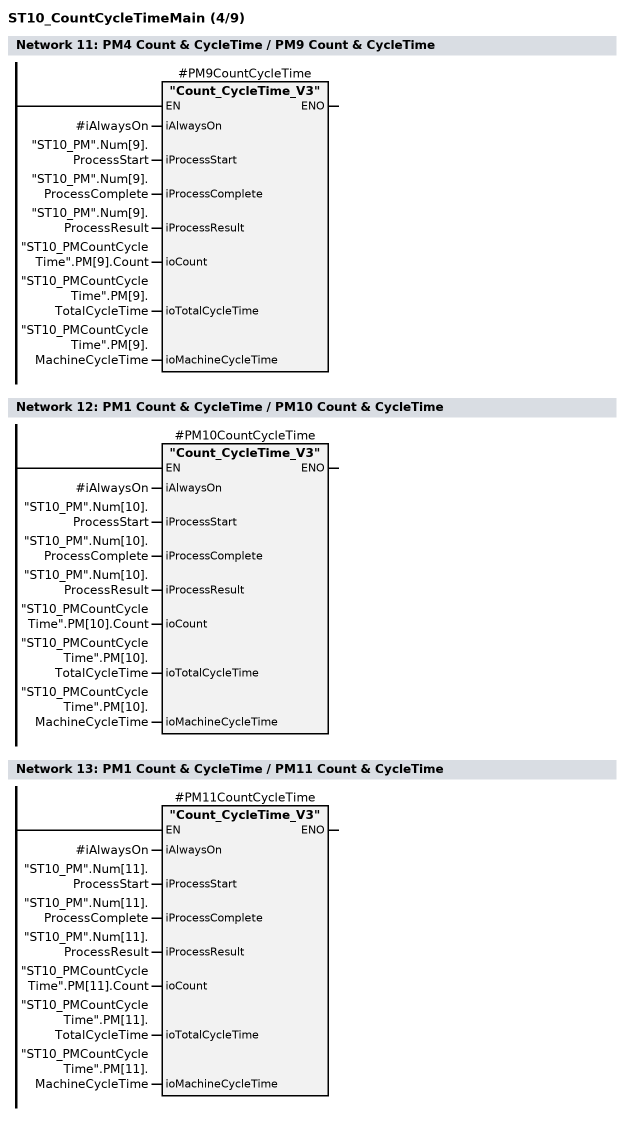
   RUNG wire#powerrail
      #PM9CountCycleTime(iAlwaysOn := #iAlwaysOn, iProcessStart := "ST10_PM".Num[9].ProcessStart, iProcessComplete := "ST10_PM".Num[9].ProcessComplete, iProcessResult := "ST10_PM".Num[9].ProcessResult, ioCount := "ST10_PMCountCycleTime".PM[9].Count, ioTotalCycleTime := "ST10_PMCountCycleTime".PM[9].TotalCycleTime, ioMachineCycleTime := "ST10_PMCountCycleTime".PM[9].MachineCycleTime)
   END_RUNG
   // the same network as SCL:
   #PM9CountCycleTime(iAlwaysOn := #iAlwaysOn,   // "Count_CycleTime_V3"
                      iProcessStart := "ST10_PM".Num[9].ProcessStart,
                      iProcessComplete := "ST10_PM".Num[9].ProcessComplete,
                      iProcessResult := "ST10_PM".Num[9].ProcessResult,
                      ioCount := "ST10_PMCountCycleTime".PM[9].Count,
                      ioTotalCycleTime := "ST10_PMCountCycleTime".PM[9].TotalCycleTime,
                      ioMachineCycleTime := "ST10_PMCountCycleTime".PM[9].MachineCycleTime);
END_REGION

REGION Network 12: PM1 Count & CycleTime / PM10 Count & CycleTime
   RUNG wire#powerrail
      #PM10CountCycleTime(iAlwaysOn := #iAlwaysOn, iProcessStart := "ST10_PM".Num[10].ProcessStart, iProcessComplete := "ST10_PM".Num[10].ProcessComplete, iProcessResult := "ST10_PM".Num[10].ProcessResult, ioCount := "ST10_PMCountCycleTime".PM[10].Count, ioTotalCycleTime := "ST10_PMCountCycleTime".PM[10].TotalCycleTime, ioMachineCycleTime := "ST10_PMCountCycleTime".PM[10].MachineCycleTime)
   END_RUNG
   // the same network as SCL:
   #PM10CountCycleTime(iAlwaysOn := #iAlwaysOn,   // "Count_CycleTime_V3"
                       iProcessStart := "ST10_PM".Num[10].ProcessStart,
                       iProcessComplete := "ST10_PM".Num[10].ProcessComplete,
                       iProcessResult := "ST10_PM".Num[10].ProcessResult,
                       ioCount := "ST10_PMCountCycleTime".PM[10].Count,
                       ioTotalCycleTime := "ST10_PMCountCycleTime".PM[10].TotalCycleTime,
                       ioMachineCycleTime := "ST10_PMCountCycleTime".PM[10].MachineCycleTime);
END_REGION

REGION Network 13: PM1 Count & CycleTime / PM11 Count & CycleTime
   RUNG wire#powerrail
      #PM11CountCycleTime(iAlwaysOn := #iAlwaysOn, iProcessStart := "ST10_PM".Num[11].ProcessStart, iProcessComplete := "ST10_PM".Num[11].ProcessComplete, iProcessResult := "ST10_PM".Num[11].ProcessResult, ioCount := "ST10_PMCountCycleTime".PM[11].Count, ioTotalCycleTime := "ST10_PMCountCycleTime".PM[11].TotalCycleTime, ioMachineCycleTime := "ST10_PMCountCycleTime".PM[11].MachineCycleTime)
   END_RUNG
   // the same network as SCL:
   #PM11CountCycleTime(iAlwaysOn := #iAlwaysOn,   // "Count_CycleTime_V3"
                       iProcessStart := "ST10_PM".Num[11].ProcessStart,
                       iProcessComplete := "ST10_PM".Num[11].ProcessComplete,
                       iProcessResult := "ST10_PM".Num[11].ProcessResult,
                       ioCount := "ST10_PMCountCycleTime".PM[11].Count,
                       ioTotalCycleTime := "ST10_PMCountCycleTime".PM[11].TotalCycleTime,
                       ioMachineCycleTime := "ST10_PMCountCycleTime".PM[11].MachineCycleTime);
END_REGION

REGION Network 14: PM1 Count & CycleTime / PM12 Count & CycleTime
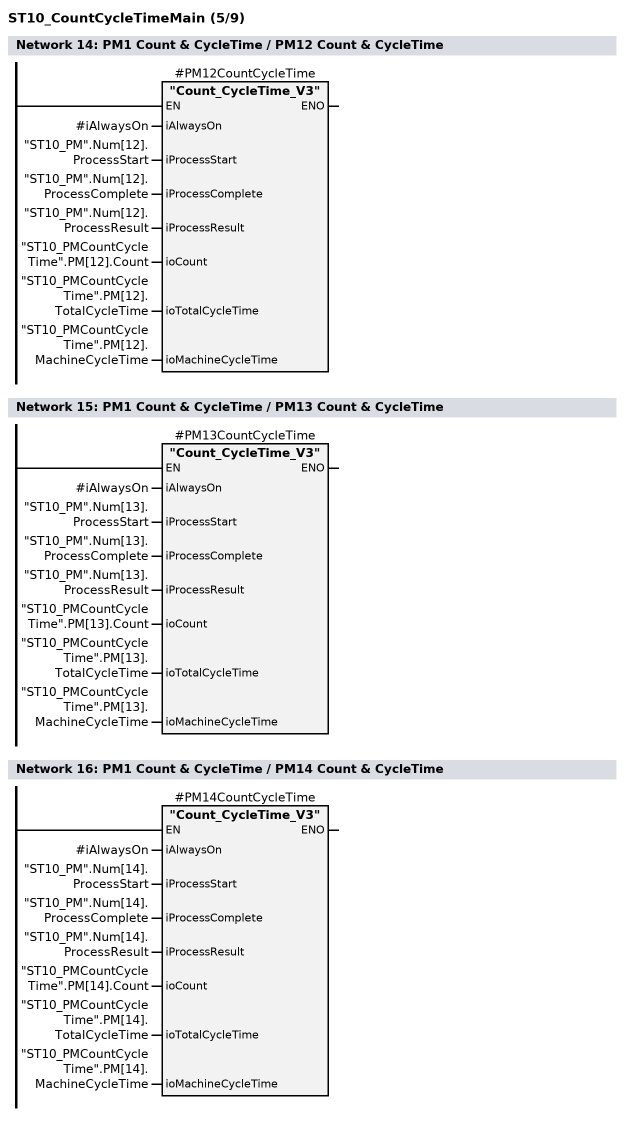
   RUNG wire#powerrail
      #PM12CountCycleTime(iAlwaysOn := #iAlwaysOn, iProcessStart := "ST10_PM".Num[12].ProcessStart, iProcessComplete := "ST10_PM".Num[12].ProcessComplete, iProcessResult := "ST10_PM".Num[12].ProcessResult, ioCount := "ST10_PMCountCycleTime".PM[12].Count, ioTotalCycleTime := "ST10_PMCountCycleTime".PM[12].TotalCycleTime, ioMachineCycleTime := "ST10_PMCountCycleTime".PM[12].MachineCycleTime)
   END_RUNG
   // the same network as SCL:
   #PM12CountCycleTime(iAlwaysOn := #iAlwaysOn,   // "Count_CycleTime_V3"
                       iProcessStart := "ST10_PM".Num[12].ProcessStart,
                       iProcessComplete := "ST10_PM".Num[12].ProcessComplete,
                       iProcessResult := "ST10_PM".Num[12].ProcessResult,
                       ioCount := "ST10_PMCountCycleTime".PM[12].Count,
                       ioTotalCycleTime := "ST10_PMCountCycleTime".PM[12].TotalCycleTime,
                       ioMachineCycleTime := "ST10_PMCountCycleTime".PM[12].MachineCycleTime);
END_REGION

REGION Network 15: PM1 Count & CycleTime / PM13 Count & CycleTime
   RUNG wire#powerrail
      #PM13CountCycleTime(iAlwaysOn := #iAlwaysOn, iProcessStart := "ST10_PM".Num[13].ProcessStart, iProcessComplete := "ST10_PM".Num[13].ProcessComplete, iProcessResult := "ST10_PM".Num[13].ProcessResult, ioCount := "ST10_PMCountCycleTime".PM[13].Count, ioTotalCycleTime := "ST10_PMCountCycleTime".PM[13].TotalCycleTime, ioMachineCycleTime := "ST10_PMCountCycleTime".PM[13].MachineCycleTime)
   END_RUNG
   // the same network as SCL:
   #PM13CountCycleTime(iAlwaysOn := #iAlwaysOn,   // "Count_CycleTime_V3"
                       iProcessStart := "ST10_PM".Num[13].ProcessStart,
                       iProcessComplete := "ST10_PM".Num[13].ProcessComplete,
                       iProcessResult := "ST10_PM".Num[13].ProcessResult,
                       ioCount := "ST10_PMCountCycleTime".PM[13].Count,
                       ioTotalCycleTime := "ST10_PMCountCycleTime".PM[13].TotalCycleTime,
                       ioMachineCycleTime := "ST10_PMCountCycleTime".PM[13].MachineCycleTime);
END_REGION

REGION Network 16: PM1 Count & CycleTime / PM14 Count & CycleTime
   RUNG wire#powerrail
      #PM14CountCycleTime(iAlwaysOn := #iAlwaysOn, iProcessStart := "ST10_PM".Num[14].ProcessStart, iProcessComplete := "ST10_PM".Num[14].ProcessComplete, iProcessResult := "ST10_PM".Num[14].ProcessResult, ioCount := "ST10_PMCountCycleTime".PM[14].Count, ioTotalCycleTime := "ST10_PMCountCycleTime".PM[14].TotalCycleTime, ioMachineCycleTime := "ST10_PMCountCycleTime".PM[14].MachineCycleTime)
   END_RUNG
   // the same network as SCL:
   #PM14CountCycleTime(iAlwaysOn := #iAlwaysOn,   // "Count_CycleTime_V3"
                       iProcessStart := "ST10_PM".Num[14].ProcessStart,
                       iProcessComplete := "ST10_PM".Num[14].ProcessComplete,
                       iProcessResult := "ST10_PM".Num[14].ProcessResult,
                       ioCount := "ST10_PMCountCycleTime".PM[14].Count,
                       ioTotalCycleTime := "ST10_PMCountCycleTime".PM[14].TotalCycleTime,
                       ioMachineCycleTime := "ST10_PMCountCycleTime".PM[14].MachineCycleTime);
END_REGION

REGION Network 17: PM1 Count & CycleTime / PM15 Count & CycleTime
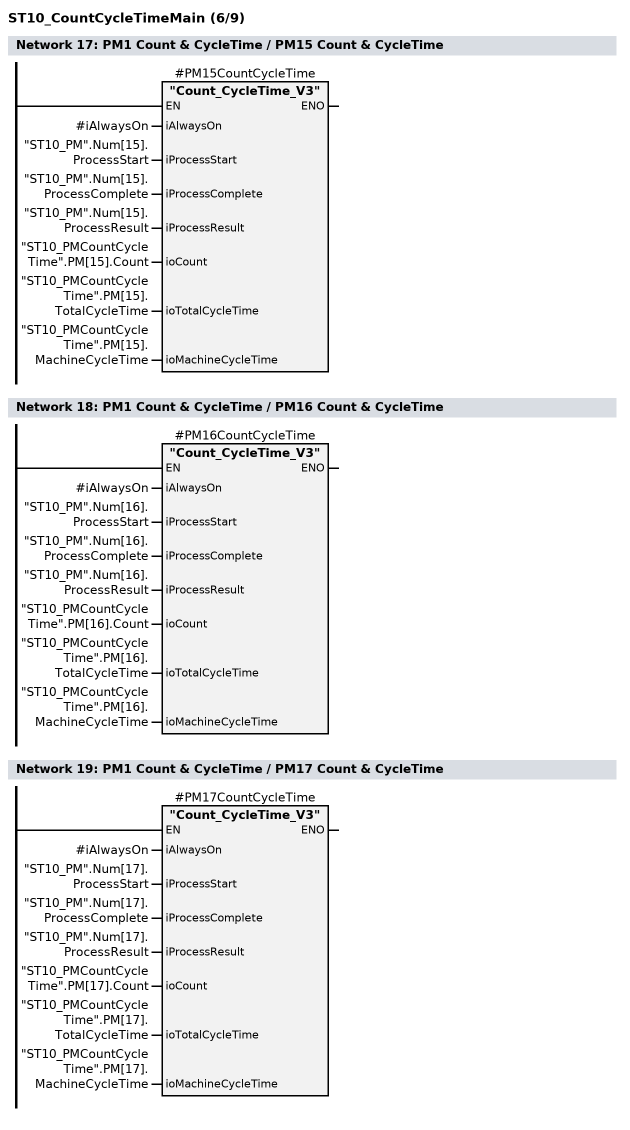
   RUNG wire#powerrail
      #PM15CountCycleTime(iAlwaysOn := #iAlwaysOn, iProcessStart := "ST10_PM".Num[15].ProcessStart, iProcessComplete := "ST10_PM".Num[15].ProcessComplete, iProcessResult := "ST10_PM".Num[15].ProcessResult, ioCount := "ST10_PMCountCycleTime".PM[15].Count, ioTotalCycleTime := "ST10_PMCountCycleTime".PM[15].TotalCycleTime, ioMachineCycleTime := "ST10_PMCountCycleTime".PM[15].MachineCycleTime)
   END_RUNG
   // the same network as SCL:
   #PM15CountCycleTime(iAlwaysOn := #iAlwaysOn,   // "Count_CycleTime_V3"
                       iProcessStart := "ST10_PM".Num[15].ProcessStart,
                       iProcessComplete := "ST10_PM".Num[15].ProcessComplete,
                       iProcessResult := "ST10_PM".Num[15].ProcessResult,
                       ioCount := "ST10_PMCountCycleTime".PM[15].Count,
                       ioTotalCycleTime := "ST10_PMCountCycleTime".PM[15].TotalCycleTime,
                       ioMachineCycleTime := "ST10_PMCountCycleTime".PM[15].MachineCycleTime);
END_REGION

REGION Network 18: PM1 Count & CycleTime / PM16 Count & CycleTime
   RUNG wire#powerrail
      #PM16CountCycleTime(iAlwaysOn := #iAlwaysOn, iProcessStart := "ST10_PM".Num[16].ProcessStart, iProcessComplete := "ST10_PM".Num[16].ProcessComplete, iProcessResult := "ST10_PM".Num[16].ProcessResult, ioCount := "ST10_PMCountCycleTime".PM[16].Count, ioTotalCycleTime := "ST10_PMCountCycleTime".PM[16].TotalCycleTime, ioMachineCycleTime := "ST10_PMCountCycleTime".PM[16].MachineCycleTime)
   END_RUNG
   // the same network as SCL:
   #PM16CountCycleTime(iAlwaysOn := #iAlwaysOn,   // "Count_CycleTime_V3"
                       iProcessStart := "ST10_PM".Num[16].ProcessStart,
                       iProcessComplete := "ST10_PM".Num[16].ProcessComplete,
                       iProcessResult := "ST10_PM".Num[16].ProcessResult,
                       ioCount := "ST10_PMCountCycleTime".PM[16].Count,
                       ioTotalCycleTime := "ST10_PMCountCycleTime".PM[16].TotalCycleTime,
                       ioMachineCycleTime := "ST10_PMCountCycleTime".PM[16].MachineCycleTime);
END_REGION

REGION Network 19: PM1 Count & CycleTime / PM17 Count & CycleTime
   RUNG wire#powerrail
      #PM17CountCycleTime(iAlwaysOn := #iAlwaysOn, iProcessStart := "ST10_PM".Num[17].ProcessStart, iProcessComplete := "ST10_PM".Num[17].ProcessComplete, iProcessResult := "ST10_PM".Num[17].ProcessResult, ioCount := "ST10_PMCountCycleTime".PM[17].Count, ioTotalCycleTime := "ST10_PMCountCycleTime".PM[17].TotalCycleTime, ioMachineCycleTime := "ST10_PMCountCycleTime".PM[17].MachineCycleTime)
   END_RUNG
   // the same network as SCL:
   #PM17CountCycleTime(iAlwaysOn := #iAlwaysOn,   // "Count_CycleTime_V3"
                       iProcessStart := "ST10_PM".Num[17].ProcessStart,
                       iProcessComplete := "ST10_PM".Num[17].ProcessComplete,
                       iProcessResult := "ST10_PM".Num[17].ProcessResult,
                       ioCount := "ST10_PMCountCycleTime".PM[17].Count,
                       ioTotalCycleTime := "ST10_PMCountCycleTime".PM[17].TotalCycleTime,
                       ioMachineCycleTime := "ST10_PMCountCycleTime".PM[17].MachineCycleTime);
END_REGION

REGION Network 20: PM1 Count & CycleTime / PM18 Count & CycleTime
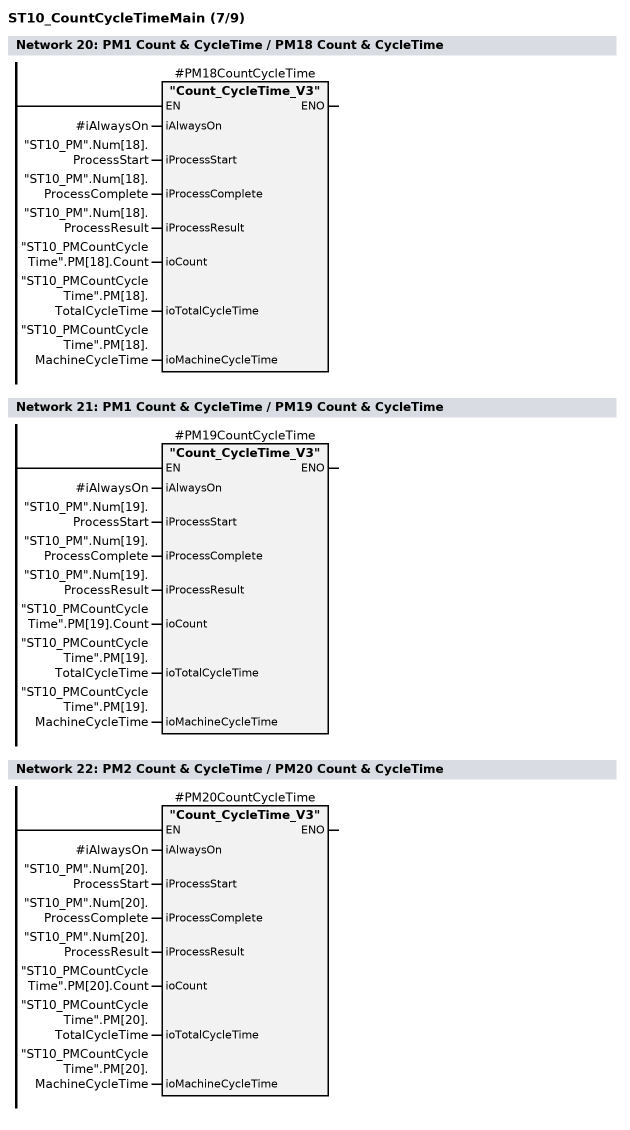
   RUNG wire#powerrail
      #PM18CountCycleTime(iAlwaysOn := #iAlwaysOn, iProcessStart := "ST10_PM".Num[18].ProcessStart, iProcessComplete := "ST10_PM".Num[18].ProcessComplete, iProcessResult := "ST10_PM".Num[18].ProcessResult, ioCount := "ST10_PMCountCycleTime".PM[18].Count, ioTotalCycleTime := "ST10_PMCountCycleTime".PM[18].TotalCycleTime, ioMachineCycleTime := "ST10_PMCountCycleTime".PM[18].MachineCycleTime)
   END_RUNG
   // the same network as SCL:
   #PM18CountCycleTime(iAlwaysOn := #iAlwaysOn,   // "Count_CycleTime_V3"
                       iProcessStart := "ST10_PM".Num[18].ProcessStart,
                       iProcessComplete := "ST10_PM".Num[18].ProcessComplete,
                       iProcessResult := "ST10_PM".Num[18].ProcessResult,
                       ioCount := "ST10_PMCountCycleTime".PM[18].Count,
                       ioTotalCycleTime := "ST10_PMCountCycleTime".PM[18].TotalCycleTime,
                       ioMachineCycleTime := "ST10_PMCountCycleTime".PM[18].MachineCycleTime);
END_REGION

